KUKA KRL program: MyProgram_296().src

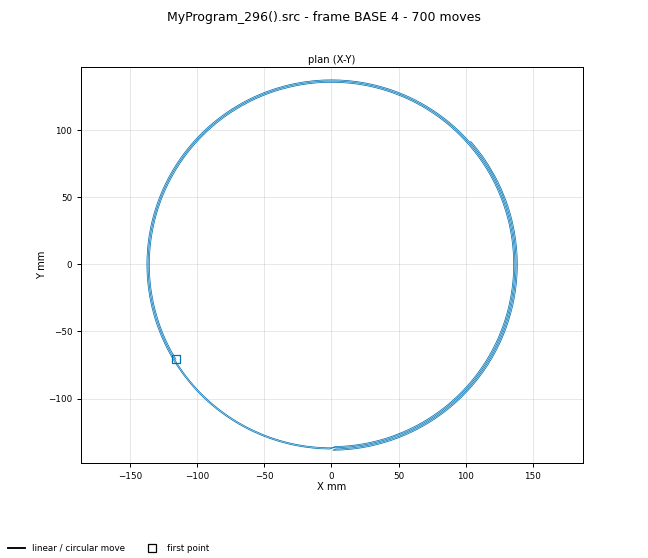
[picture p0: tool path of MyProgram_296().src in frame BASE 4, 700 of 700 moves have a stored position in this frame; points joined in program order, loops and branches not executed]
&ACCESS RVP
&REL 1
&PARAM TEMPLATE = C:\KRC\Roboter\Template\vorgabe
&PARAM EDITMASK = *
DEF MyProgram_296()
; ---- Setting reference (Base) ----
$BASE = BASE_DATA[4]

; --------------------------
; ---- Setting tool (TCP) ----
$TOOL = TOOL_DATA[3]
; --------------------------

$VEL.CP = VEL_APROX_PRINT
Startdeposition()
$VEL.CP = VEL_PRINT
LIN {X -116.0636,Y -70.6635,Z 178,A -146.1492,B 6.2959,C 0.3309,E1 6.1676,E2 238.3864} C_DIS
LIN {X -119.6803,Y -64.347,Z 178,A -149.1984,B 6.2963,C 0.3231,E1 6.1634,E2 241.4316} C_DIS
LIN {X -121.2417,Y -61.3507,Z 178,A -150.649,B 6.2965,C 0.3198,E1 6.1615,E2 242.8846} C_DIS
LIN {X -123.4162,Y -56.8493,Z 178,A -152.7977,B 6.2967,C 0.3149,E1 6.159,E2 245.0373} C_DIS
LIN {X -124.8313,Y -53.6711,Z 178,A -154.2629,B 6.2969,C 0.3111,E1 6.1573,E2 246.5015} C_DIS
LIN {X -126.1562,Y -50.4788,Z 178,A -155.7795,B 6.2971,C 0.3079,E1 6.1557,E2 248.0246} C_DIS
LIN {X -127.9876,Y -45.6377,Z 178,A -158.0309,B 6.2973,C 0.3029,E1 6.1535,E2 250.2832} C_DIS
LIN {X -129.1495,Y -42.2414,Z 178,A -159.6948,B 6.2974,C 0.3004,E1 6.152,E2 251.9649} C_DIS
LIN {X -131.3967,Y -34.6191,Z 178,A -163.2762,B 6.2978,C 0.2937,E1 6.1493,E2 255.5726} C_DIS
LIN {X -132.2272,Y -31.3001,Z 178,A -164.3938,B 6.2981,C 0.2863,E1 6.1486,E2 256.649} C_DIS
LIN {X -132.8516,Y -28.5293,Z 178,A -165.6891,B 6.2981,C 0.284,E1 6.1478,E2 257.9556} C_DIS
LIN {X -133.5646,Y -24.9844,Z 178,A -167.1822,B 6.2984,C 0.2794,E1 6.147,E2 259.4438} C_DIS
LIN {X -134.0652,Y -22.1367,Z 178,A -168.5264,B 6.2984,C 0.2773,E1 6.1464,E2 260.8025} C_DIS
LIN {X -134.7069,Y -17.8196,Z 178,A -170.3512,B 6.2987,C 0.2719,E1 6.1457,E2 262.6241} C_DIS
LIN {X -135.1168,Y -14.3862,Z 178,A -171.8433,B 6.2989,C 0.2681,E1 6.1452,E2 264.1192} C_DIS
LIN {X -135.4888,Y -10.3173,Z 178,A -173.6674,B 6.299,C 0.2643,E1 6.1448,E2 265.9546} C_DIS
LIN {X -135.7321,Y -6.3646,Z 178,A -175.3605,B 6.2992,C 0.2598,E1 6.1445,E2 267.6493} C_DIS
LIN {X -135.8577,Y -2.5014,Z 178,A -176.9735,B 6.2994,C 0.2549,E1 6.1444,E2 269.2588} C_DIS
LIN {X -135.8765,Y 1.1885,Z 178,A -178.6131,B 6.2996,C 0.2514,E1 6.1444,E2 270.9075} C_DIS
LIN {X -135.7799,Y 5.2289,Z 178,A 179.6851,B 6.2998,C 0.2464,E1 6.1445,E2 272.6076} C_DIS
LIN {X -135.6091,Y 8.5868,Z 178,A 178.1279,B 6.2998,C 0.2438,E1 6.1448,E2 274.1807} C_DIS
LIN {X -135.2372,Y 13.2071,Z 178,A 176.2276,B 6.3001,C 0.2377,E1 6.1453,E2 276.0728} C_DIS
LIN {X -134.7736,Y 17.3106,Z 178,A 174.3999,B 6.3003,C 0.2337,E1 6.1459,E2 277.9096} C_DIS
LIN {X -134.2648,Y 20.8907,Z 178,A 172.9,B 6.3004,C 0.2291,E1 6.1465,E2 279.4051} C_DIS
LIN {X -133.7038,Y 24.2246,Z 178,A 171.44,B 6.3006,C 0.2254,E1 6.1472,E2 280.8681} C_DIS
LIN {X -133.1263,Y 27.2185,Z 178,A 170.1483,B 6.3006,C 0.2218,E1 6.1479,E2 282.1594} C_DIS
LIN {X -132.3925,Y 30.5906,Z 178,A 168.6598,B 6.3008,C 0.2181,E1 6.1488,E2 283.6507} C_DIS
LIN {X -131.5728,Y 33.9457,Z 178,A 166.9358,B 6.3008,C 0.2169,E1 6.15,E2 285.4061} C_DIS
LIN {X -130.369,Y 38.3059,Z 178,A 165.1776,B 6.3011,C 0.21,E1 6.1513,E2 287.1444} C_DIS
LIN {X -129.3497,Y 41.619,Z 178,A 163.4434,B 6.3011,C 0.2089,E1 6.1528,E2 288.9105} C_DIS
LIN {X -127.4729,Y 47.0581,Z 178,A 161.2834,B 6.3014,C 0.1995,E1 6.1548,E2 291.036} C_DIS
LIN {X -125.8737,Y 51.1795,Z 178,A 159.3113,B 6.3015,C 0.1957,E1 6.1568,E2 293.0195} C_DIS
LIN {X -124.4446,Y 54.5655,Z 178,A 157.5921,B 6.3016,C 0.1934,E1 6.1587,E2 294.7579} C_DIS
LIN {X -123.226,Y 57.2606,Z 178,A 156.3891,B 6.3017,C 0.1897,E1 6.1601,E2 295.9544} C_DIS
LIN {X -121.8373,Y 60.1584,Z 178,A 154.3031,B 6.3016,C 0.1939,E1 6.1628,E2 298.1274} C_DIS
LIN {X -119.1995,Y 65.2335,Z 178,A 152.7848,B 6.3021,C 0.1784,E1 6.1647,E2 299.5357} C_DIS
LIN {X -117.7028,Y 67.897,Z 178,A 150.9757,B 6.302,C 0.1807,E1 6.1673,E2 301.4067} C_DIS
LIN {X -116.0163,Y 70.7408,Z 178,A 150.0425,B 6.3022,C 0.1724,E1 6.1685,E2 302.2829} C_DIS
LIN {X -112.7627,Y 75.8199,Z 178,A 147.1337,B 6.3022,C 0.1702,E1 6.173,E2 305.2338} C_DIS
LIN {X -110.1908,Y 79.5109,Z 178,A 145.2766,B 6.3024,C 0.1653,E1 6.176,E2 307.0844} C_DIS
LIN {X -107.6516,Y 82.9169,Z 178,A 143.3645,B 6.3024,C 0.1625,E1 6.1792,E2 309.0094} C_DIS
LIN {X -104.8415,Y 86.4421,Z 178,A 141.4392,B 6.3026,C 0.1586,E1 6.1826,E2 310.9359} C_DIS
LIN {X -101.8749,Y 89.9189,Z 178,A 139.5339,B 6.3026,C 0.1542,E1 6.1861,E2 312.8368} C_DIS
LIN {X -99.0063,Y 93.0683,Z 178,A 137.6552,B 6.3028,C 0.1513,E1 6.1897,E2 314.7239} C_DIS
LIN {X -95.9062,Y 96.2598,Z 178,A 135.7647,B 6.3028,C 0.1476,E1 6.1934,E2 316.6145} C_DIS
LIN {X -92.7534,Y 99.3014,Z 178,A 133.8742,B 6.3029,C 0.1445,E1 6.1972,E2 318.5085} C_DIS
LIN {X -89.3426,Y 102.3806,Z 178,A 131.9344,B 6.303,C 0.1408,E1 6.2013,E2 320.447} C_DIS
LIN {X -85.8899,Y 105.2941,Z 178,A 130.0021,B 6.303,C 0.1377,E1 6.2054,E2 322.3809} C_DIS
LIN {X -82.27,Y 108.1465,Z 178,A 128.0373,B 6.3031,C 0.1345,E1 6.2098,E2 324.3468} C_DIS
LIN {X -78.7448,Y 110.7397,Z 178,A 126.1286,B 6.3031,C 0.1322,E1 6.2141,E2 326.2615} C_DIS
LIN {X -74.9969,Y 113.3114,Z 178,A 123.4447,B 6.3031,C 0.1379,E1 6.2206,E2 329.0355} C_DIS
LIN {X -69.7447,Y 116.6175,Z 178,A 121.7746,B 6.3034,C 0.1231,E1 6.2243,E2 330.5904} C_DIS
LIN {X -66.8937,Y 118.2763,Z 178,A 120.1144,B 6.3034,C 0.1243,E1 6.2284,E2 332.2819} C_DIS
LIN {X -63.0682,Y 120.3568,Z 178,A 118.3471,B 6.3034,C 0.121,E1 6.2327,E2 334.0395} C_DIS
LIN {X -59.8342,Y 121.9972,Z 178,A 116.798,B 6.3034,C 0.1193,E1 6.2366,E2 335.5899} C_DIS
LIN {X -55.8012,Y 123.894,Z 178,A 114.9346,B 6.3034,C 0.1169,E1 6.2413,E2 337.45} C_DIS
LIN {X -52.2464,Y 125.434,Z 178,A 113.2307,B 6.3035,C 0.116,E1 6.2457,E2 339.1611} C_DIS
LIN {X -47.376,Y 127.3538,Z 178,A 110.5367,B 6.3035,C 0.1196,E1 6.2529,E2 341.9118} C_DIS
LIN {X -43.1002,Y 128.8635,Z 178,A 109.4047,B 6.3036,C 0.1084,E1 6.2556,E2 342.9489} C_DIS
LIN {X -38.9004,Y 130.195,Z 178,A 107.001,B 6.3036,C 0.1136,E1 6.2622,E2 345.4171} C_DIS
LIN {X -34.4811,Y 131.4335,Z 178,A 105.3513,B 6.3036,C 0.1086,E1 6.2665,E2 347.0314} C_DIS
LIN {X -31.6898,Y 132.1333,Z 178,A 104.1647,B 6.3036,C 0.1075,E1 6.2698,E2 348.214} C_DIS
LIN {X -28.623,Y 132.8313,Z 178,A 102.7874,B 6.3036,C 0.1073,E1 6.2735,E2 349.5966} C_DIS
LIN {X -25.1145,Y 133.5398,Z 178,A 101.3076,B 6.3036,C 0.1062,E1 6.2776,E2 351.0719} C_DIS
LIN {X -22.0251,Y 134.0838,Z 178,A 99.9239,B 6.3036,C 0.1063,E1 6.2814,E2 352.4622} C_DIS
LIN {X -18.0004,Y 134.6832,Z 178,A 98.1327,B 6.3036,C 0.1066,E1 6.2864,E2 354.2616} C_DIS
LIN {X -14.1094,Y 135.1465,Z 178,A 96.5823,B 6.3037,C 0.1048,E1 6.2906,E2 355.7989} C_DIS
LIN {X -10.0268,Y 135.51,Z 178,A 94.5302,B 6.3037,C 0.1087,E1 6.2965,E2 357.8889} C_DIS
LIN {X -6.7551,Y 135.7125,Z 178,A 93.4747,B 6.3037,C 0.1042,E1 6.2993,E2 358.9046} C_DIS
LIN {X -3.2262,Y 135.8433,Z 178,A 91.4247,B 6.3036,C 0.1115,E1 6.3052,E2 361.0211} C_DIS
LIN {X 1.2847,Y 135.8755,Z 178,A 89.9059,B 6.3036,C 0.1065,E1 6.3093,E2 362.4932} C_DIS
LIN {X 5.7731,Y 135.7586,Z 178,A 88.2731,B 6.3037,C 0.1033,E1 6.3138,E2 364.0939} C_DIS
LIN {X 8.3573,Y 135.6232,Z 178,A 87.0566,B 6.3037,C 0.1052,E1 6.3172,E2 365.3251} C_DIS
LIN {X 14.3269,Y 135.1231,Z 178,A 84.6214,B 6.3037,C 0.1046,E1 6.324,E2 367.7485} C_DIS
LIN {X 17.5541,Y 134.7417,Z 178,A 83.1449,B 6.3037,C 0.1066,E1 6.3281,E2 369.2373} C_DIS
LIN {X 20.9839,Y 134.2504,Z 178,A 81.677,B 6.3037,C 0.1073,E1 6.3321,E2 370.7055} C_DIS
LIN {X 25.3585,Y 133.4931,Z 178,A 79.7741,B 6.3037,C 0.1087,E1 6.3374,E2 372.6116} C_DIS
LIN {X 28.8609,Y 132.78,Z 178,A 78.3733,B 6.3037,C 0.1082,E1 6.3412,E2 373.9992} C_DIS
LIN {X 32.1612,Y 132.0196,Z 178,A 76.9512,B 6.3037,C 0.1091,E1 6.345,E2 375.4201} C_DIS
LIN {X 36.1084,Y 130.9956,Z 178,A 74.6656,B 6.3035,C 0.1184,E1 6.3514,E2 377.7734} C_DIS
LIN {X 40.7031,Y 129.6422,Z 178,A 73.2942,B 6.3035,C 0.1109,E1 6.3548,E2 379.0665} C_DIS
LIN {X 44.6522,Y 128.3339,Z 178,A 71.4391,B 6.3035,C 0.114,E1 6.3598,E2 380.9335} C_DIS
LIN {X 48.3697,Y 126.9816,Z 178,A 69.8436,B 6.3035,C 0.1146,E1 6.3639,E2 382.52} C_DIS
LIN {X 50.941,Y 125.9699,Z 178,A 68.6824,B 6.3035,C 0.1158,E1 6.3669,E2 383.6806} C_DIS
LIN {X 53.9208,Y 124.7234,Z 178,A 67.3009,B 6.3035,C 0.1176,E1 6.3705,E2 385.0643} C_DIS
LIN {X 57.2157,Y 123.2468,Z 178,A 65.8286,B 6.3035,C 0.1187,E1 6.3742,E2 386.5304} C_DIS
LIN {X 60.5933,Y 121.6227,Z 178,A 64.2467,B 6.3035,C 0.1208,E1 6.3782,E2 388.1125} C_DIS
LIN {X 64.1271,Y 119.7985,Z 178,A 62.4843,B 6.3033,C 0.1243,E1 6.3826,E2 389.8853} C_DIS
LIN {X 68.2573,Y 117.4942,Z 178,A 60.5431,B 6.3033,C 0.1263,E1 6.3873,E2 391.82} C_DIS
LIN {X 71.8437,Y 115.336,Z 178,A 58.82,B 6.3033,C 0.1284,E1 6.3914,E2 393.5381} C_DIS
LIN {X 76.4158,Y 112.3593,Z 178,A 56.6264,B 6.3033,C 0.1304,E1 6.3965,E2 395.7189} C_DIS
LIN {X 79.5335,Y 110.1744,Z 178,A 54.9237,B 6.3031,C 0.1346,E1 6.4004,E2 397.4336} C_DIS
LIN {X 83.0535,Y 107.5457,Z 178,A 53.1981,B 6.3031,C 0.1358,E1 6.4042,E2 399.144} C_DIS
LIN {X 86.2241,Y 105.021,Z 178,A 51.4142,B 6.3031,C 0.1401,E1 6.4081,E2 400.9372} C_DIS
LIN {X 89.6033,Y 102.1531,Z 178,A 49.6048,B 6.303,C 0.1426,E1 6.4119,E2 402.7398} C_DIS
LIN {X 95.2128,Y 96.9455,Z 178,A 46.5727,B 6.3029,C 0.1459,E1 6.418,E2 405.7488} C_DIS
LIN {X 99.6056,Y 92.4266,Z 178,A 43.7905,B 6.3027,C 0.1534,E1 6.4234,E2 408.547} C_DIS
LIN {X 102.5276,Y 89.1742,Z 178,A 41.9627,B 6.3027,C 0.1571,E1 6.4268,E2 410.3735} C_DIS
LIN {X 106.7379,Y 84.089,Z 178,A 39.465,B 6.3026,C 0.1587,E1 6.4312,E2 412.8371} C_DIS
LIN {X 108.7546,Y 81.4646,Z 178,A 37.8869,B 6.3024,C 0.1648,E1 6.4338,E2 414.4381} C_DIS
LIN {X 111.1727,Y 78.1318,Z 178,A 36.1359,B 6.3024,C 0.1691,E1 6.4367,E2 416.1915} C_DIS
LIN {X 113.7751,Y 74.2917,Z 178,A 34.241,B 6.3022,C 0.1727,E1 6.4396,E2 418.0797} C_DIS
LIN {X 116.1679,Y 70.491,Z 178,A 32.382,B 6.3022,C 0.1768,E1 6.4423,E2 419.9353} C_DIS
LIN {X 118.4324,Y 66.6159,Z 178,A 30.5441,B 6.302,C 0.1806,E1 6.4449,E2 421.7674} C_DIS
LIN {X 120.3327,Y 63.1142,Z 178,A 28.9081,B 6.3019,C 0.1841,E1 6.447,E2 423.3988} C_DIS
LIN {X 121.9972,Y 59.8342,Z 178,A 27.4637,B 6.3019,C 0.1863,E1 6.4488,E2 424.8309} C_DIS
LIN {X 123.6119,Y 56.4261,Z 178,A 25.7789,B 6.3017,C 0.192,E1 6.4508,E2 426.5282} C_DIS
LIN {X 126.4203,Y 49.8165,Z 178,A 23.0232,B 6.3016,C 0.1955,E1 6.4538,E2 429.252} C_DIS
LIN {X 128.0463,Y 45.4749,Z 178,A 21.0403,B 6.3014,C 0.2012,E1 6.4557,E2 431.2396} C_DIS
LIN {X 129.0556,Y 42.5232,Z 178,A 19.7314,B 6.3013,C 0.2046,E1 6.4568,E2 432.5485} C_DIS
LIN {X 129.9574,Y 39.6798,Z 178,A 18.5302,B 6.3012,C 0.2071,E1 6.4578,E2 433.7435} C_DIS
LIN {X 130.813,Y 36.7614,Z 178,A 17.2145,B 6.301,C 0.2112,E1 6.4588,E2 435.0641} C_DIS
LIN {X 131.6892,Y 33.4868,Z 178,A 15.8447,B 6.301,C 0.2141,E1 6.4598,E2 436.4274} C_DIS
LIN {X 132.6532,Y 29.4479,Z 178,A 14.0247,B 6.3007,C 0.2202,E1 6.4609,E2 438.2572} C_DIS
LIN {X 133.4336,Y 25.67,Z 178,A 12.5388,B 6.3007,C 0.2224,E1 6.4617,E2 439.7268} C_DIS
LIN {X 134.0567,Y 22.1875,Z 178,A 11.1081,B 6.3005,C 0.2255,E1 6.4624,E2 441.151} C_DIS
LIN {X 134.6366,Y 18.3559,Z 178,A 9.3768,B 6.3003,C 0.2318,E1 6.4631,E2 442.8956} C_DIS
LIN {X 135.129,Y 14.2725,Z 178,A 7.7678,B 6.3003,C 0.2346,E1 6.4636,E2 444.4903} C_DIS
LIN {X 135.5055,Y 10.0889,Z 178,A 5.5412,B 6.2997,C 0.2473,E1 6.4641,E2 446.7746} C_DIS
LIN {X 135.7694,Y 5.496,Z 178,A 3.6419,B 6.2995,C 0.2521,E1 6.4643,E2 448.6705} C_DIS
LIN {X 135.8783,Y 0.862,Z 178,A 2.2313,B 6.2997,C 0.2487,E1 6.4643,E2 450.0152} C_DIS
LIN {X 135.8374,Y -3.4376,Z 178,A -0.0974,B 6.2991,C 0.2625,E1 6.4643,E2 452.4093} C_DIS
LIN {X 135.6249,Y -8.3298,Z 178,A -1.5744,B 6.2993,C 0.2585,E1 6.464,E2 453.815} C_DIS
LIN {X 135.3457,Y -12.0589,Z 178,A -3.0356,B 6.2992,C 0.2611,E1 6.4637,E2 455.2633} C_DIS
LIN {X 134.9715,Y -15.6945,Z 178,A -4.6162,B 6.299,C 0.2662,E1 6.4632,E2 456.85} C_DIS
LIN {X 134.5126,Y -19.2305,Z 178,A -6.0496,B 6.2988,C 0.2693,E1 6.4627,E2 458.276} C_DIS
LIN {X 133.7779,Y -23.8102,Z 178,A -7.9361,B 6.2987,C 0.2736,E1 6.4618,E2 460.1554} C_DIS
LIN {X 133.1003,Y -27.3461,Z 178,A -9.4108,B 6.2985,C 0.2772,E1 6.461,E2 461.6261} C_DIS
LIN {X 132.4098,Y -30.5147,Z 178,A -10.7699,B 6.2983,C 0.2809,E1 6.4602,E2 462.9853} C_DIS
LIN {X 131.0461,Y -35.9279,Z 178,A -13.0212,B 6.2981,C 0.2858,E1 6.4586,E2 465.2259} C_DIS
LIN {X 130.2592,Y -38.6811,Z 178,A -14.2667,B 6.2979,C 0.2897,E1 6.4576,E2 466.4773} C_DIS
LIN {X 129.4087,Y -41.4344,Z 178,A -15.4712,B 6.2978,C 0.2929,E1 6.4566,E2 467.6816} C_DIS
LIN {X 127.5161,Y -46.9427,Z 178,A -17.8777,B 6.2975,C 0.2988,E1 6.4544,E2 470.0842} C_DIS
LIN {X 125.5505,Y -51.9675,Z 178,A -19.9244,B 6.2975,C 0.3011,E1 6.4523,E2 472.1041} C_DIS
LIN {X 124.5223,Y -54.3858,Z 178,A -21.2164,B 6.2971,C 0.3071,E1 6.4509,E2 473.4204} C_DIS
LIN {X 122.7582,Y -58.2572,Z 178,A -23.0205,B 6.2969,C 0.312,E1 6.4488,E2 475.2274} C_DIS
LIN {X 120.4896,Y -62.8153,Z 178,A -24.9253,B 6.2969,C 0.3135,E1 6.4464,E2 477.1037} C_DIS
LIN {X 119.1979,Y -65.2366,Z 178,A -26.2432,B 6.2965,C 0.3191,E1 6.4446,E2 478.443} C_DIS
LIN {X 116.9538,Y -69.18,Z 178,A -28.1146,B 6.2963,C 0.3233,E1 6.442,E2 480.311} C_DIS
LIN {X 114.814,Y -72.6751,Z 178,A -29.7899,B 6.2961,C 0.3267,E1 6.4395,E2 481.9811} C_DIS
LIN {X 112.3358,Y -76.4506,Z 178,A -31.681,B 6.2959,C 0.3311,E1 6.4366,E2 483.8724} C_DIS
LIN {X 109.8749,Y -79.9467,Z 178,A -33.4551,B 6.2957,C 0.3349,E1 6.4337,E2 485.6446} C_DIS
LIN {X 107.3491,Y -83.3071,Z 178,A -35.1877,B 6.2955,C 0.3384,E1 6.4308,E2 487.3737} C_DIS
LIN {X 104.5102,Y -86.8422,Z 178,A -37.0651,B 6.2953,C 0.3422,E1 6.4275,E2 489.2486} C_DIS
LIN {X 101.6631,Y -90.1586,Z 178,A -38.8818,B 6.2951,C 0.3459,E1 6.4241,E2 491.0636} C_DIS
LIN {X 98.6198,Y -93.478,Z 178,A -40.7569,B 6.2949,C 0.3496,E1 6.4206,E2 492.9374} C_DIS
LIN {X 95.4318,Y -96.7308,Z 178,A -43.1438,B 6.2943,C 0.3611,E1 6.4157,E2 495.3849} C_DIS
LIN {X 91.8687,Y -100.1198,Z 178,A -44.5572,B 6.2946,C 0.3547,E1 6.413,E2 496.7168} C_DIS
LIN {X 89.5658,Y -102.1859,Z 178,A -45.8294,B 6.2946,C 0.3568,E1 6.4104,E2 497.9861} C_DIS
LIN {X 86.7428,Y -104.5925,Z 178,A -47.5068,B 6.2942,C 0.3616,E1 6.4067,E2 499.6792} C_DIS
LIN {X 83.086,Y -107.5205,Z 178,A -49.4306,B 6.2941,C 0.3644,E1 6.4025,E2 501.5982} C_DIS
LIN {X 79.6611,Y -110.0819,Z 178,A -51.2109,B 6.2939,C 0.3673,E1 6.3985,E2 503.377} C_DIS
LIN {X 76.2647,Y -112.4616,Z 178,A -52.9478,B 6.2937,C 0.3701,E1 6.3945,E2 505.114} C_DIS
LIN {X 72.5451,Y -114.8961,Z 178,A -54.8077,B 6.2936,C 0.3729,E1 6.3902,E2 506.9736} C_DIS
LIN {X 68.5178,Y -117.3429,Z 178,A -56.7639,B 6.2934,C 0.3756,E1 6.3855,E2 508.9275} C_DIS
LIN {X 64.7472,Y -119.4648,Z 178,A -58.5983,B 6.2932,C 0.3784,E1 6.381,E2 510.7646} C_DIS
LIN {X 60.8473,Y -121.4974,Z 178,A -60.5263,B 6.293,C 0.3822,E1 6.3762,E2 512.7035} C_DIS
LIN {X 56.7439,Y -123.4649,Z 178,A -62.1933,B 6.2931,C 0.3808,E1 6.372,E2 514.3399} C_DIS
LIN {X 53.9979,Y -124.69,Z 178,A -63.73,B 6.2928,C 0.3865,E1 6.368,E2 515.9116} C_DIS
LIN {X 46.4657,Y -127.689,Z 178,A -66.7659,B 6.2928,C 0.3846,E1 6.3602,E2 518.9015} C_DIS
LIN {X 41.9034,Y -129.2588,Z 178,A -68.7651,B 6.2928,C 0.3862,E1 6.3549,E2 520.8976} C_DIS
LIN {X 38.4539,Y -130.3257,Z 178,A -70.4167,B 6.2926,C 0.3896,E1 6.3505,E2 522.5667} C_DIS
LIN {X 34.8173,Y -131.3439,Z 178,A -71.9768,B 6.2926,C 0.3905,E1 6.3463,E2 524.1237} C_DIS
LIN {X 31.4044,Y -132.2021,Z 178,A -73.3966,B 6.2925,C 0.3907,E1 6.3424,E2 525.5364} C_DIS
LIN {X 28.2597,Y -132.9098,Z 178,A -74.9104,B 6.2923,C 0.394,E1 6.3383,E2 527.0707} C_DIS
LIN {X 24.0792,Y -133.7298,Z 178,A -76.8012,B 6.2921,C 0.3965,E1 6.333,E2 528.9745} C_DIS
LIN {X 18.4191,Y -134.6284,Z 178,A -78.9444,B 6.2923,C 0.3939,E1 6.3272,E2 531.0846} C_DIS
LIN {X 15.1531,Y -135.0342,Z 178,A -81.1475,B 6.2915,C 0.4061,E1 6.3208,E2 533.3915} C_DIS
LIN {X 9.2312,Y -135.5681,Z 178,A -82.7583,B 6.2923,C 0.3943,E1 6.3166,E2 534.8903} C_DIS
LIN {X 2.4002,Y -135.8594,Z 178,A -85.6824,B 6.2922,C 0.3955,E1 6.3085,E2 537.8211} C_DIS
LIN {X 2.4002,Y -135.8594,Z 178,A -85.6824,B 6.2922,C 0.3955,E1 6.3085,E2 537.8212} C_DIS
Enddeposition()
LIN {X 0.9937,Y -136.781,Z 178,A -85.9393,B 6.2292,C 0.3941,E1 6.2447,E2 538.0864} C_DIS
Startdeposition()
$VEL.CP = VEL_PRINT
LIN {X 7.0143,Y -136.6048,Z 178,A -83.1394,B 6.2294,C 0.3897,E1 6.2526,E2 535.2495} C_DIS
LIN {X 13.8862,Y -136.08,Z 178,A -80.1066,B 6.2296,C 0.3865,E1 6.2611,E2 532.1964} C_DIS
LIN {X 22.8856,Y -134.857,Z 178,A -76.3832,B 6.2296,C 0.3857,E1 6.2714,E2 528.4815} C_DIS
LIN {X 26.6198,Y -134.1709,Z 178,A -74.7602,B 6.2298,C 0.3842,E1 6.2758,E2 526.8533} C_DIS
LIN {X 30.257,Y -133.3962,Z 178,A -73.3123,B 6.2298,C 0.3847,E1 6.2797,E2 525.4186} C_DIS
LIN {X 33.2653,Y -132.6783,Z 178,A -71.9723,B 6.2298,C 0.383,E1 6.2834,E2 524.072} C_DIS
LIN {X 37.0999,Y -131.6573,Z 178,A -70.408,B 6.2298,C 0.383,E1 6.2876,E2 522.5193} C_DIS
LIN {X 40.7775,Y -130.5671,Z 178,A -68.7967,B 6.2299,C 0.3814,E1 6.2919,E2 520.9063} C_DIS
LIN {X 43.894,Y -129.5522,Z 178,A -67.2601,B 6.2302,C 0.3775,E1 6.296,E2 519.3475} C_DIS
LIN {X 53.8396,Y -125.7436,Z 178,A -63.1247,B 6.2302,C 0.3775,E1 6.3067,E2 515.2513} C_DIS
LIN {X 58.4249,Y -123.6802,Z 178,A -61.0159,B 6.2304,C 0.3747,E1 6.312,E2 513.1408} C_DIS
LIN {X 61.008,Y -122.4265,Z 178,A -59.7426,B 6.2305,C 0.3719,E1 6.3153,E2 511.8574} C_DIS
LIN {X 64.4799,Y -120.6354,Z 178,A -57.9955,B 6.2308,C 0.3678,E1 6.3196,E2 510.0947} C_DIS
LIN {X 68.4273,Y -118.4406,Z 178,A -56.1417,B 6.2308,C 0.3656,E1 6.3241,E2 508.2443} C_DIS
LIN {X 72.5143,Y -115.9837,Z 178,A -54.1992,B 6.231,C 0.3633,E1 6.3287,E2 506.3072} C_DIS
LIN {X 76.1478,Y -113.6311,Z 178,A -52.4262,B 6.2312,C 0.3609,E1 6.3328,E2 504.538} C_DIS
LIN {X 79.823,Y -111.0804,Z 178,A -50.5401,B 6.2314,C 0.3574,E1 6.3372,E2 502.6487} C_DIS
LIN {X 83.246,Y -108.5385,Z 178,A -48.8043,B 6.2314,C 0.355,E1 6.341,E2 500.9178} C_DIS
LIN {X 86.8047,Y -105.7143,Z 178,A -46.9088,B 6.2317,C 0.3516,E1 6.3451,E2 499.0216} C_DIS
LIN {X 91.8683,Y -101.3444,Z 178,A -43.8168,B 6.2323,C 0.3413,E1 6.3517,E2 495.8894} C_DIS
LIN {X 94.8582,Y -98.552,Z 178,A -42.3552,B 6.2323,C 0.3419,E1 6.3546,E2 494.4592} C_DIS
LIN {X 98.5146,Y -94.897,Z 178,A -40.3012,B 6.2323,C 0.3392,E1 6.3586,E2 492.4177} C_DIS
LIN {X 101.6106,Y -91.5747,Z 178,A -38.4541,B 6.2326,C 0.3359,E1 6.362,E2 490.576} C_DIS
LIN {X 104.4722,Y -88.2959,Z 178,A -36.6477,B 6.2328,C 0.3321,E1 6.3653,E2 488.77} C_DIS
LIN {X 107.3567,Y -84.765,Z 178,A -34.7947,B 6.2329,C 0.3287,E1 6.3685,E2 486.9226} C_DIS
LIN {X 109.9748,Y -81.3399,Z 178,A -33.0306,B 6.2331,C 0.3252,E1 6.3715,E2 485.1622} C_DIS
LIN {X 112.4928,Y -77.8201,Z 178,A -31.2377,B 6.2333,C 0.3211,E1 6.3744,E2 483.3703} C_DIS
LIN {X 114.9924,Y -74.0767,Z 178,A -29.3673,B 6.2336,C 0.3168,E1 6.3772,E2 481.5} C_DIS
LIN {X 117.4366,Y -70.1364,Z 178,A -27.5436,B 6.2336,C 0.3139,E1 6.3799,E2 479.6897} C_DIS
LIN {X 119.4847,Y -66.5884,Z 178,A -25.963,B 6.2338,C 0.3119,E1 6.382,E2 478.1251} C_DIS
LIN {X 121.8235,Y -62.2011,Z 178,A -23.8208,B 6.2341,C 0.3055,E1 6.3848,E2 475.9732} C_DIS
LIN {X 123.4477,Y -58.9116,Z 178,A -22.2217,B 6.2344,C 0.3004,E1 6.3868,E2 474.3646} C_DIS
LIN {X 125.4043,Y -54.6243,Z 178,A -20.512,B 6.2344,C 0.2997,E1 6.3887,E2 472.6871} C_DIS
LIN {X 126.7997,Y -51.3009,Z 178,A -19.122,B 6.2344,C 0.2976,E1 6.3902,E2 471.311} C_DIS
LIN {X 127.9897,Y -48.2561,Z 178,A -17.6236,B 6.2348,C 0.2918,E1 6.3917,E2 469.7949} C_DIS
LIN {X 129.3482,Y -44.4871,Z 178,A -16.0266,B 6.2349,C 0.2886,E1 6.3932,E2 468.2067} C_DIS
LIN {X 130.4059,Y -41.284,Z 178,A -14.586,B 6.2351,C 0.2842,E1 6.3944,E2 466.7613} C_DIS
LIN {X 131.3176,Y -38.284,Z 178,A -13.3802,B 6.2351,C 0.2824,E1 6.3954,E2 465.5681} C_DIS
LIN {X 132.0354,Y -35.7334,Z 178,A -12.3491,B 6.2353,C 0.2807,E1 6.3961,E2 464.5461} C_DIS
LIN {X 132.8418,Y -32.6091,Z 178,A -10.9141,B 6.2355,C 0.2755,E1 6.3971,E2 463.0993} C_DIS
LIN {X 133.6585,Y -29.0765,Z 178,A -9.3989,B 6.2357,C 0.2713,E1 6.398,E2 461.5831} C_DIS
LIN {X 134.3139,Y -25.8806,Z 178,A -8.0398,B 6.2358,C 0.2675,E1 6.3988,E2 460.2238} C_DIS
LIN {X 134.9897,Y -22.0897,Z 178,A -6.4213,B 6.236,C 0.2629,E1 6.3995,E2 458.6032} C_DIS
LIN {X 135.5908,Y -18.0342,Z 178,A -4.811,B 6.2362,C 0.2598,E1 6.4001,E2 457.0051} C_DIS
LIN {X 136.0879,Y -13.8085,Z 178,A -2.5856,B 6.2367,C 0.2472,E1 6.4008,E2 454.7215} C_DIS
LIN {X 136.4609,Y -9.4217,Z 178,A -0.6421,B 6.237,C 0.2402,E1 6.4012,E2 452.7637} C_DIS
LIN {X 136.7206,Y -4.2081,Z 178,A 0.9836,B 6.2368,C 0.2435,E1 6.4013,E2 451.2081} C_DIS
LIN {X 136.7815,Y -1.0613,Z 178,A 2.9325,B 6.2374,C 0.229,E1 6.4013,E2 449.1773} C_DIS
LIN {X 136.6944,Y 4.9829,Z 178,A 4.802,B 6.2372,C 0.2331,E1 6.4013,E2 447.3908} C_DIS
LIN {X 136.3411,Y 11.0178,Z 178,A 7.1487,B 6.2374,C 0.229,E1 6.4008,E2 445.0659} C_DIS
LIN {X 135.7969,Y 16.4097,Z 178,A 9.3818,B 6.2376,C 0.2232,E1 6.4001,E2 442.8357} C_DIS
LIN {X 135.2647,Y 20.3425,Z 178,A 10.8423,B 6.2376,C 0.2219,E1 6.3995,E2 441.3996} C_DIS
LIN {X 134.696,Y 23.8134,Z 178,A 12.3983,B 6.2378,C 0.2163,E1 6.3988,E2 439.8321} C_DIS
LIN {X 134.0427,Y 27.2495,Z 178,A 13.7971,B 6.2379,C 0.2133,E1 6.398,E2 438.4406} C_DIS
LIN {X 133.423,Y 30.1393,Z 178,A 14.9502,B 6.238,C 0.2113,E1 6.3974,E2 437.2974} C_DIS
LIN {X 132.7895,Y 32.8261,Z 178,A 16.2855,B 6.2382,C 0.2051,E1 6.3965,E2 435.9388} C_DIS
LIN {X 131.8515,Y 36.4054,Z 178,A 17.7044,B 6.2382,C 0.203,E1 6.3954,E2 434.5354} C_DIS
LIN {X 130.8627,Y 39.8115,Z 178,A 18.9442,B 6.2382,C 0.203,E1 6.3945,E2 433.3256} C_DIS
LIN {X 129.8964,Y 42.8604,Z 178,A 20.4036,B 6.2385,C 0.1974,E1 6.3932,E2 431.8503} C_DIS
LIN {X 128.8212,Y 45.9916,Z 178,A 21.8189,B 6.2385,C 0.1932,E1 6.3919,E2 430.4306} C_DIS
LIN {X 127.7315,Y 48.9392,Z 178,A 23.0076,B 6.2386,C 0.1918,E1 6.3907,E2 429.2572} C_DIS
LIN {X 126.476,Y 52.0979,Z 178,A 24.731,B 6.2389,C 0.1831,E1 6.3889,E2 427.4953} C_DIS
LIN {X 125.2112,Y 55.0709,Z 178,A 25.9385,B 6.2389,C 0.182,E1 6.3876,E2 426.3055} C_DIS
LIN {X 123.6218,Y 58.5471,Z 178,A 27.4571,B 6.239,C 0.1792,E1 6.3858,E2 424.7963} C_DIS
LIN {X 122.0165,Y 61.8218,Z 178,A 28.8945,B 6.239,C 0.1768,E1 6.384,E2 423.3695} C_DIS
LIN {X 120.2231,Y 65.2454,Z 178,A 30.5035,B 6.2392,C 0.1729,E1 6.3819,E2 421.761} C_DIS
LIN {X 118.211,Y 68.824,Z 178,A 32.2071,B 6.2392,C 0.1689,E1 6.3795,E2 420.0586} C_DIS
LIN {X 115.9754,Y 72.5277,Z 178,A 34.0126,B 6.2394,C 0.1646,E1 6.3769,E2 418.2531} C_DIS
LIN {X 113.5789,Y 76.226,Z 178,A 35.8177,B 6.2394,C 0.1609,E1 6.3741,E2 416.4524} C_DIS
LIN {X 111.0987,Y 79.7974,Z 178,A 37.6117,B 6.2396,C 0.1571,E1 6.3712,E2 414.6611} C_DIS
LIN {X 108.6744,Y 83.0683,Z 178,A 39.242,B 6.2396,C 0.1544,E1 6.3685,E2 413.0396} C_DIS
LIN {X 106.5603,Y 85.7635,Z 178,A 40.7585,B 6.2398,C 0.1499,E1 6.3658,E2 411.5123} C_DIS
LIN {X 103.3768,Y 89.5759,Z 178,A 42.7564,B 6.2398,C 0.1467,E1 6.3622,E2 409.5242} C_DIS
LIN {X 100.5575,Y 92.7292,Z 178,A 44.6373,B 6.24,C 0.1412,E1 6.3586,E2 407.6291} C_DIS
LIN {X 96.7471,Y 96.6986,Z 178,A 46.7218,B 6.24,C 0.1399,E1 6.3546,E2 405.5716} C_DIS
LIN {X 92.7195,Y 100.5663,Z 178,A 49.0276,B 6.24,C 0.1359,E1 6.35,E2 403.2694} C_DIS
LIN {X 89.4084,Y 103.5212,Z 178,A 50.8664,B 6.2402,C 0.1327,E1 6.3461,E2 401.4328} C_DIS
LIN {X 86.0779,Y 106.3068,Z 178,A 52.6024,B 6.2402,C 0.1306,E1 6.3424,E2 399.7068} C_DIS
LIN {X 82.8994,Y 108.8035,Z 178,A 54.3427,B 6.2402,C 0.1269,E1 6.3385,E2 397.9604} C_DIS
LIN {X 79.5471,Y 111.2777,Z 178,A 56.0168,B 6.2403,C 0.1251,E1 6.3348,E2 396.2949} C_DIS
LIN {X 76.0397,Y 113.7033,Z 178,A 57.8094,B 6.2403,C 0.1221,E1 6.3306,E2 394.5014} C_DIS
LIN {X 72.2393,Y 116.1548,Z 178,A 59.6747,B 6.2404,C 0.1196,E1 6.3262,E2 392.6396} C_DIS
LIN {X 68.3691,Y 118.4743,Z 178,A 61.5347,B 6.2404,C 0.1173,E1 6.3217,E2 390.7833} C_DIS
LIN {X 64.5467,Y 120.5995,Z 178,A 63.3359,B 6.2405,C 0.1152,E1 6.3173,E2 388.9859} C_DIS
LIN {X 61.2122,Y 122.3257,Z 178,A 64.799,B 6.2405,C 0.1148,E1 6.3137,E2 387.5364} C_DIS
LIN {X 57.849,Y 123.9502,Z 178,A 66.4324,B 6.2405,C 0.1119,E1 6.3096,E2 385.8946} C_DIS
LIN {X 54.465,Y 125.4732,Z 178,A 67.911,B 6.2405,C 0.1111,E1 6.3058,E2 384.4254} C_DIS
LIN {X 51.309,Y 126.7965,Z 178,A 69.2894,B 6.2405,C 0.1104,E1 6.3023,E2 383.054} C_DIS
LIN {X 48.619,Y 127.8538,Z 178,A 70.4732,B 6.2406,C 0.1095,E1 6.2992,E2 381.8737} C_DIS
LIN {X 45.2143,Y 129.0961,Z 178,A 72.0325,B 6.2406,C 0.1074,E1 6.2951,E2 380.3096} C_DIS
LIN {X 42.2972,Y 130.0823,Z 178,A 73.4587,B 6.2406,C 0.1043,E1 6.2913,E2 378.8668} C_DIS
LIN {X 37.8153,Y 131.4548,Z 178,A 75.4038,B 6.2407,C 0.1029,E1 6.2861,E2 376.9243} C_DIS
LIN {X 33.6513,Y 132.5804,Z 178,A 77.1027,B 6.2407,C 0.1031,E1 6.2815,E2 375.2391} C_DIS
LIN {X 29.6954,Y 133.5244,Z 178,A 78.7725,B 6.2407,C 0.1024,E1 6.277,E2 373.574} C_DIS
LIN {X 25.8451,Y 134.3207,Z 178,A 80.416,B 6.2407,C 0.1015,E1 6.2725,E2 371.9313} C_DIS
LIN {X 22.4458,Y 134.9303,Z 178,A 81.8522,B 6.2407,C 0.1009,E1 6.2685,E2 370.4969} C_DIS
LIN {X 18.702,Y 135.5016,Z 178,A 83.7273,B 6.2408,C 0.0963,E1 6.2633,E2 368.5867} C_DIS
LIN {X 15.3526,Y 135.9222,Z 178,A 85.2227,B 6.2408,C 0.0946,E1 6.2591,E2 367.0817} C_DIS
LIN {X 11.697,Y 136.2837,Z 178,A 86.5157,B 6.2408,C 0.0976,E1 6.2556,E2 365.8196} C_DIS
LIN {X 8.0217,Y 136.5498,Z 178,A 88.4945,B 6.2408,C 0.0914,E1 6.2499,E2 363.7876} C_DIS
LIN {X 3.1021,Y 136.7513,Z 178,A 89.9166,B 6.2408,C 0.0998,E1 6.2462,E2 362.4455} C_DIS
LIN {X -3.9297,Y 136.7283,Z 178,A 92.8771,B 6.2408,C 0.0997,E1 6.2379,E2 359.4846} C_DIS
LIN {X -6.5681,Y 136.6272,Z 178,A 94.6736,B 6.2409,C 0.0906,E1 6.2327,E2 357.6035} C_DIS
LIN {X -11.7409,Y 136.28,Z 178,A 96.1523,B 6.2408,C 0.1002,E1 6.2288,E2 356.2114} C_DIS
LIN {X -15.1734,Y 135.9415,Z 178,A 97.6966,B 6.2408,C 0.0993,E1 6.2244,E2 354.6557} C_DIS
LIN {X -19.1134,Y 135.4428,Z 178,A 99.3372,B 6.2408,C 0.1002,E1 6.2199,E2 353.0189} C_DIS
LIN {X -22.0645,Y 134.994,Z 178,A 100.4539,B 6.2408,C 0.1025,E1 6.2169,E2 351.9192} C_DIS
LIN {X -25.578,Y 134.3718,Z 178,A 102.0512,B 6.2408,C 0.1019,E1 6.2125,E2 350.3102} C_DIS
LIN {X -28.4393,Y 133.7961,Z 178,A 103.263,B 6.2408,C 0.1027,E1 6.2091,E2 349.1005} C_DIS
LIN {X -31.8302,Y 133.0296,Z 178,A 104.7985,B 6.2408,C 0.1027,E1 6.2049,E2 347.5561} C_DIS
LIN {X -35.2494,Y 132.1645,Z 178,A 106.2329,B 6.2407,C 0.1042,E1 6.2011,E2 346.1279} C_DIS
LIN {X -38.7487,Y 131.1816,Z 178,A 107.7775,B 6.2407,C 0.1051,E1 6.1969,E2 344.5816} C_DIS
LIN {X -42.5857,Y 129.9879,Z 178,A 109.4039,B 6.2407,C 0.1072,E1 6.1926,E2 342.9633} C_DIS
LIN {X -48.8812,Y 127.754,Z 178,A 112.3044,B 6.2407,C 0.1087,E1 6.185,E2 340.0523} C_DIS
LIN {X -53.8752,Y 125.7282,Z 178,A 114.5788,B 6.2406,C 0.1109,E1 6.1791,E2 337.7774} C_DIS
LIN {X -57.0897,Y 124.3012,Z 178,A 116.0319,B 6.2406,C 0.1128,E1 6.1754,E2 336.3278} C_DIS
LIN {X -59.6197,Y 123.1094,Z 178,A 117.22,B 6.2406,C 0.114,E1 6.1724,E2 335.1386} C_DIS
LIN {X -62.5654,Y 121.638,Z 178,A 118.7491,B 6.2406,C 0.114,E1 6.1686,E2 333.5922} C_DIS
LIN {X -66.6785,Y 119.4345,Z 178,A 120.7509,B 6.2405,C 0.1161,E1 6.1637,E2 331.5861} C_DIS
LIN {X -70.6221,Y 117.1453,Z 178,A 122.4027,B 6.2404,C 0.1219,E1 6.1598,E2 329.9675} C_DIS
LIN {X -74.0479,Y 115.0109,Z 178,A 124.3574,B 6.2404,C 0.1214,E1 6.1551,E2 327.9817} C_DIS
LIN {X -77.6386,Y 112.6179,Z 178,A 126.1934,B 6.2404,C 0.1239,E1 6.1508,E2 326.1437} C_DIS
LIN {X -81.3667,Y 109.9549,Z 178,A 128.1314,B 6.2403,C 0.1269,E1 6.1464,E2 324.205} C_DIS
LIN {X -84.8917,Y 107.2567,Z 178,A 130.0542,B 6.2403,C 0.1295,E1 6.1422,E2 322.2759} C_DIS
LIN {X -88.4302,Y 104.358,Z 178,A 131.9804,B 6.2402,C 0.1328,E1 6.1381,E2 320.3501} C_DIS
LIN {X -91.519,Y 101.6604,Z 178,A 133.7044,B 6.2401,C 0.136,E1 6.1345,E2 318.6268} C_DIS
LIN {X -94.6574,Y 98.7445,Z 178,A 135.5235,B 6.2401,C 0.1393,E1 6.1308,E2 316.8062} C_DIS
LIN {X -97.8767,Y 95.5547,Z 178,A 137.4689,B 6.2399,C 0.1426,E1 6.1269,E2 314.8567} C_DIS
LIN {X -100.9463,Y 92.3062,Z 178,A 139.4094,B 6.2399,C 0.1457,E1 6.1232,E2 312.9094} C_DIS
LIN {X -103.9386,Y 88.9236,Z 178,A 141.34,B 6.2398,C 0.1494,E1 6.1197,E2 310.9757} C_DIS
LIN {X -106.8754,Y 85.3708,Z 178,A 143.2818,B 6.2397,C 0.1536,E1 6.1163,E2 309.0342} C_DIS
LIN {X -109.6543,Y 81.7704,Z 178,A 145.1547,B 6.2396,C 0.1583,E1 6.1131,E2 307.167} C_DIS
LIN {X -112.0886,Y 78.401,Z 178,A 147.0064,B 6.2395,C 0.1611,E1 6.1101,E2 305.3032} C_DIS
LIN {X -113.7953,Y 75.9018,Z 178,A 148.3277,B 6.2395,C 0.1635,E1 6.1081,E2 303.9765} C_DIS
LIN {X -116.995,Y 70.8706,Z 178,A 150.7809,B 6.2393,C 0.1701,E1 6.1044,E2 301.5311} C_DIS
LIN {X -119.1541,Y 67.1773,Z 178,A 152.6196,B 6.2391,C 0.1741,E1 6.1019,E2 299.6882} C_DIS
LIN {X -120.8566,Y 64.0613,Z 178,A 154.4391,B 6.2391,C 0.1742,E1 6.0994,E2 297.8287} C_DIS
LIN {X -122.5022,Y 60.8543,Z 178,A 155.4993,B 6.2389,C 0.1829,E1 6.0982,E2 296.8257} C_DIS
LIN {X -123.7079,Y 58.367,Z 178,A 156.7886,B 6.2389,C 0.1845,E1 6.0966,E2 295.5213} C_DIS
LIN {X -125.3432,Y 54.7656,Z 178,A 158.5391,B 6.2387,C 0.1879,E1 6.0946,E2 293.7606} C_DIS
LIN {X -126.5992,Y 51.7985,Z 178,A 159.8141,B 6.2387,C 0.1922,E1 6.0932,E2 292.4961} C_DIS
LIN {X -127.9131,Y 48.4607,Z 178,A 161.2753,B 6.2385,C 0.1967,E1 6.0918,E2 291.0414} C_DIS
LIN {X -130.2347,Y 41.8201,Z 178,A 164.3784,B 6.2383,C 0.203,E1 6.089,E2 287.9217} C_DIS
LIN {X -131.9797,Y 35.9422,Z 178,A 166.9968,B 6.2381,C 0.2096,E1 6.0869,E2 285.2994} C_DIS
LIN {X -132.8936,Y 32.3943,Z 178,A 168.6591,B 6.238,C 0.2125,E1 6.0858,E2 283.6226} C_DIS
LIN {X -133.6839,Y 28.9586,Z 178,A 170.0332,B 6.2378,C 0.2177,E1 6.0849,E2 282.2626} C_DIS
LIN {X -134.2239,Y 26.3515,Z 178,A 171.4147,B 6.2378,C 0.2181,E1 6.0842,E2 280.8489} C_DIS
LIN {X -135.0172,Y 21.925,Z 178,A 173.3235,B 6.2376,C 0.2231,E1 6.0833,E2 278.9386} C_DIS
LIN {X -135.598,Y 17.9788,Z 178,A 174.9217,B 6.2374,C 0.2286,E1 6.0827,E2 277.3508} C_DIS
LIN {X -136.0136,Y 14.5032,Z 178,A 176.4892,B 6.2373,C 0.2317,E1 6.0822,E2 275.7718} C_DIS
LIN {X -136.3665,Y 10.7137,Z 178,A 178.2316,B 6.2372,C 0.2347,E1 6.0818,E2 274.0123} C_DIS
LIN {X -136.6496,Y 6.1225,Z 178,A -179.858,B 6.237,C 0.2404,E1 6.0815,E2 272.1056} C_DIS
LIN {X -136.7672,Y 2.1942,Z 178,A -178.2559,B 6.2368,C 0.2456,E1 6.0814,E2 270.5103} C_DIS
LIN {X -136.7725,Y -1.8726,Z 178,A -176.6504,B 6.2365,C 0.2515,E1 6.0814,E2 268.9184} C_DIS
LIN {X -136.676,Y -5.4545,Z 178,A -174.9356,B 6.2365,C 0.2535,E1 6.0816,E2 267.178} C_DIS
LIN {X -136.4421,Y -9.6792,Z 178,A -173.2043,B 6.2362,C 0.259,E1 6.0819,E2 265.4531} C_DIS
LIN {X -136.1497,Y -13.1643,Z 178,A -171.6589,B 6.2361,C 0.2623,E1 6.0823,E2 263.8987} C_DIS
LIN {X -135.7191,Y -17.0552,Z 178,A -169.8919,B 6.2359,C 0.2656,E1 6.0828,E2 262.117} C_DIS
LIN {X -135.1763,Y -20.9137,Z 178,A -168.3506,B 6.2357,C 0.2712,E1 6.0835,E2 260.5883} C_DIS
LIN {X -134.6008,Y -24.345,Z 178,A -166.8199,B 6.2356,C 0.2745,E1 6.0842,E2 259.0494} C_DIS
LIN {X -133.7975,Y -28.4328,Z 178,A -165.1869,B 6.2353,C 0.2805,E1 6.0851,E2 257.4317} C_DIS
LIN {X -133.0693,Y -31.6653,Z 178,A -163.5422,B 6.2353,C 0.2816,E1 6.0862,E2 255.7555} C_DIS
LIN {X -130.8679,Y -39.7945,Z 178,A -160.062,B 6.2348,C 0.2918,E1 6.0888,E2 252.2838} C_DIS
LIN {X -129.6789,Y -43.5137,Z 178,A -157.8108,B 6.2348,C 0.2895,E1 6.0908,E2 249.9554} C_DIS
LIN {X -128.1288,Y -47.8847,Z 178,A -156.4749,B 6.2343,C 0.3013,E1 6.092,E2 248.6979} C_DIS
LIN {X -127.1483,Y -50.4361,Z 178,A -155.2531,B 6.2343,C 0.3035,E1 6.0933,E2 247.467} C_DIS
LIN {X -125.6947,Y -53.9528,Z 178,A -153.5692,B 6.2341,C 0.3067,E1 6.0951,E2 245.7725} C_DIS
LIN {X -124.3042,Y -57.0833,Z 178,A -152.0708,B 6.2339,C 0.3097,E1 6.0969,E2 244.2668} C_DIS
LIN {X -122.496,Y -60.867,Z 178,A -150.3038,B 6.2337,C 0.314,E1 6.099,E2 242.4994} C_DIS
LIN {X -120.4756,Y -64.7773,Z 178,A -148.4031,B 6.2335,C 0.318,E1 6.1015,E2 240.5925} C_DIS
LIN {X -118.1137,Y -68.9909,Z 178,A -146.2502,B 6.2333,C 0.3215,E1 6.1045,E2 238.4241} C_DIS
LIN {X -115.7426,Y -72.8981,Z 178,A -144.367,B 6.2331,C 0.3264,E1 6.1073,E2 236.5457} C_DIS
LIN {X -113.243,Y -76.7235,Z 178,A -142.3815,B 6.2329,C 0.33,E1 6.1103,E2 234.5518} C_DIS
LIN {X -110.5695,Y -80.5291,Z 178,A -140.5964,B 6.2325,C 0.3363,E1 6.1132,E2 232.7884} C_DIS
LIN {X -108.2177,Y -83.6626,Z 178,A -138.7385,B 6.2325,C 0.3375,E1 6.1164,E2 230.9033} C_DIS
LIN {X -105.5435,Y -87.0122,Z 178,A -136.8625,B 6.2323,C 0.3404,E1 6.1197,E2 229.0177} C_DIS
LIN {X -102.6501,Y -90.4073,Z 178,A -134.5418,B 6.2323,C 0.3391,E1 6.1241,E2 226.6393} C_DIS
LIN {X -99.5507,Y -93.809,Z 178,A -133.0379,B 6.2319,C 0.3479,E1 6.1269,E2 225.1905} C_DIS
LIN {X -97.2525,Y -96.1899,Z 178,A -131.6169,B 6.2318,C 0.3502,E1 6.1296,E2 223.7654} C_DIS
LIN {X -94.1487,Y -99.2302,Z 178,A -129.7763,B 6.2316,C 0.3535,E1 6.1333,E2 221.9225} C_DIS
LIN {X -90.9159,Y -102.2004,Z 178,A -127.869,B 6.2314,C 0.356,E1 6.1373,E2 220.0069} C_DIS
LIN {X -87.6867,Y -104.9838,Z 178,A -126.0865,B 6.2313,C 0.3592,E1 6.1411,E2 218.2251} C_DIS
LIN {X -84.1434,Y -107.845,Z 178,A -124.1493,B 6.2311,C 0.3621,E1 6.1454,E2 216.2844} C_DIS
LIN {X -80.8573,Y -110.3294,Z 178,A -122.4746,B 6.2309,C 0.3655,E1 6.1491,E2 214.6163} C_DIS
LIN {X -77.2899,Y -112.8572,Z 178,A -120.5672,B 6.2308,C 0.3674,E1 6.1535,E2 212.6993} C_DIS
LIN {X -73.5506,Y -115.3292,Z 178,A -118.7325,B 6.2306,C 0.3707,E1 6.1578,E2 210.8702} C_DIS
LIN {X -70.1207,Y -117.446,Z 178,A -116.9537,B 6.2306,C 0.3719,E1 6.1621,E2 209.0798} C_DIS
LIN {X -66.1746,Y -119.7138,Z 178,A -115.0682,B 6.2304,C 0.3747,E1 6.1666,E2 207.1969} C_DIS
LIN {X -62.3866,Y -121.729,Z 178,A -113.2249,B 6.2303,C 0.3763,E1 6.1712,E2 205.3475} C_DIS
LIN {X -59.1175,Y -123.3493,Z 178,A -111.7763,B 6.2301,C 0.379,E1 6.1748,E2 203.9091} C_DIS
LIN {X -56.0351,Y -124.7799,Z 178,A -110.3652,B 6.23,C 0.3807,E1 6.1784,E2 202.4995} C_DIS
LIN {X -53.0109,Y -126.0947,Z 178,A -109.0394,B 6.2299,C 0.3829,E1 6.1818,E2 201.1808} C_DIS
LIN {X -50.4859,Y -127.1283,Z 178,A -107.6379,B 6.2299,C 0.3806,E1 6.1855,E2 199.7457} C_DIS
LIN {X -46.7867,Y -128.5345,Z 178,A -106.2564,B 6.2297,C 0.3857,E1 6.189,E2 198.3996} C_DIS
LIN {X -43.5841,Y -129.6554,Z 178,A -104.5132,B 6.2299,C 0.3826,E1 6.1938,E2 196.6145} C_DIS
LIN {X -38.8046,Y -131.1652,Z 178,A -102.499,B 6.2297,C 0.3853,E1 6.1991,E2 194.6109} C_DIS
LIN {X -35.2878,Y -132.1542,Z 178,A -101.0651,B 6.2296,C 0.3875,E1 6.2029,E2 193.1891} C_DIS
LIN {X -32.5097,Y -132.8658,Z 178,A -99.9025,B 6.2295,C 0.3887,E1 6.2061,E2 192.0313} C_DIS
LIN {X -29.8238,Y -133.4951,Z 178,A -98.528,B 6.2296,C 0.3864,E1 6.2099,E2 190.6281} C_DIS
LIN {X -25.9115,Y -134.308,Z 178,A -96.9813,B 6.2295,C 0.3888,E1 6.2141,E2 189.0973} C_DIS
LIN {X -21.8121,Y -135.0361,Z 178,A -94.88,B 6.2298,C 0.3846,E1 6.22,E2 186.9491} C_DIS
LIN {X -18.2992,Y -135.556,Z 178,A -93.1162,B 6.23,C 0.3811,E1 6.225,E2 185.1487} C_DIS
LIN {X -13.2943,Y -136.1372,Z 178,A -91.8632,B 6.2292,C 0.3934,E1 6.2282,E2 184.0064} C_DIS
LIN {X -7.4064,Y -136.5851,Z 178,A -89.0276,B 6.2295,C 0.3886,E1 6.2362,E2 181.123} C_DIS
LIN {X -3.4054,Y -136.7429,Z 178,A -87.3786,B 6.2295,C 0.3889,E1 6.2408,E2 179.477} C_DIS
LIN {X 0.9937,Y -136.781,Z 178,A -85.937,B 6.2291,C 0.3944,E1 6.2447,E2 178.0864} C_DIS
Enddeposition()
LIN {X 0.9937,Y -136.781,Z 178,A -85.937,B 6.2291,C 0.3944,E1 6.2447,E2 178.0864} C_DIS
Startdeposition()
$VEL.CP = VEL_PRINT
LIN {X -1.1234,Y -137.6849,Z 178,A -87.0809,B 6.1678,C 0.4013,E1 6.1805,E2 179.3151} C_DIS
LIN {X -4.5941,Y -137.6145,Z 178,A -88.5059,B 6.1678,C 0.4011,E1 6.1765,E2 180.7383} C_DIS
LIN {X -7.5479,Y -137.4834,Z 178,A -89.7432,B 6.1678,C 0.4011,E1 6.173,E2 181.977} C_DIS
LIN {X -10.6641,Y -137.2768,Z 178,A -91.0339,B 6.1678,C 0.4009,E1 6.1695,E2 183.2671} C_DIS
LIN {X -13.5262,Y -137.0234,Z 178,A -92.2645,B 6.1678,C 0.4012,E1 6.166,E2 184.5026} C_DIS
LIN {X -16.9565,Y -136.6423,Z 178,A -93.687,B 6.1678,C 0.4007,E1 6.1621,E2 185.9239} C_DIS
LIN {X -20.272,Y -136.1906,Z 178,A -95.08,B 6.1678,C 0.4004,E1 6.1582,E2 187.3176} C_DIS
LIN {X -23.4576,Y -135.6782,Z 178,A -96.4293,B 6.1679,C 0.4,E1 6.1545,E2 188.6682} C_DIS
LIN {X -26.1273,Y -135.1874,Z 178,A -97.603,B 6.1679,C 0.4,E1 6.1513,E2 189.8478} C_DIS
LIN {X -29.7133,Y -134.4461,Z 178,A -99.0969,B 6.1679,C 0.399,E1 6.1472,E2 191.3383} C_DIS
LIN {X -33.0685,Y -133.6612,Z 178,A -100.5391,B 6.168,C 0.3983,E1 6.1433,E2 192.782} C_DIS
LIN {X -35.7187,Y -132.9751,Z 178,A -101.7077,B 6.168,C 0.398,E1 6.1401,E2 193.9547} C_DIS
LIN {X -39.4924,Y -131.906,Z 178,A -103.3293,B 6.1681,C 0.3967,E1 6.1358,E2 195.5753} C_DIS
LIN {X -42.7003,Y -130.9027,Z 178,A -104.7388,B 6.1681,C 0.3958,E1 6.132,E2 196.9865} C_DIS
LIN {X -45.7564,Y -129.8652,Z 178,A -106.0926,B 6.1682,C 0.3949,E1 6.1284,E2 198.342} C_DIS
LIN {X -48.948,Y -128.6961,Z 178,A -107.519,B 6.1683,C 0.3938,E1 6.1247,E2 199.7701} C_DIS
LIN {X -52.1265,Y -127.4419,Z 178,A -108.954,B 6.1683,C 0.3926,E1 6.121,E2 201.207} C_DIS
LIN {X -55.2886,Y -126.1022,Z 178,A -110.3813,B 6.1685,C 0.3911,E1 6.1173,E2 202.6343} C_DIS
LIN {X -58.0991,Y -124.8307,Z 178,A -111.7276,B 6.1685,C 0.3905,E1 6.1139,E2 203.9887} C_DIS
LIN {X -61.5503,Y -123.1672,Z 178,A -113.3094,B 6.1686,C 0.3885,E1 6.1099,E2 205.569} C_DIS
LIN {X -65.3102,Y -121.2157,Z 178,A -115.1229,B 6.1687,C 0.3869,E1 6.1054,E2 207.389} C_DIS
LIN {X -69.0449,Y -119.1279,Z 178,A -116.9405,B 6.1689,C 0.3851,E1 6.101,E2 209.2115} C_DIS
LIN {X -72.3058,Y -117.1778,Z 178,A -118.4887,B 6.169,C 0.3825,E1 6.0973,E2 210.7555} C_DIS
LIN {X -75.6352,Y -115.0564,Z 178,A -120.2378,B 6.169,C 0.3814,E1 6.0931,E2 212.5181} C_DIS
LIN {X -78.9364,Y -112.8176,Z 178,A -121.8429,B 6.1693,C 0.3782,E1 6.0895,E2 214.116} C_DIS
LIN {X -81.8762,Y -110.7029,Z 178,A -123.459,B 6.1693,C 0.3771,E1 6.0858,E2 215.746} C_DIS
LIN {X -85.3425,Y -108.053,Z 178,A -125.2979,B 6.1695,C 0.3743,E1 6.0817,E2 217.5876} C_DIS
LIN {X -88.7792,Y -105.2475,Z 178,A -127.0859,B 6.1697,C 0.3704,E1 6.0779,E2 219.368} C_DIS
LIN {X -91.8459,Y -102.5815,Z 178,A -128.8655,B 6.1699,C 0.3684,E1 6.0742,E2 221.1585} C_DIS
LIN {X -94.8096,Y -99.8498,Z 178,A -130.4982,B 6.1701,C 0.3647,E1 6.0708,E2 222.7852} C_DIS
LIN {X -97.305,Y -97.4193,Z 178,A -132.0295,B 6.1701,C 0.3629,E1 6.0678,E2 224.3267} C_DIS
LIN {X -100.4058,Y -94.2203,Z 178,A -133.8562,B 6.1704,C 0.3589,E1 6.0643,E2 226.1494} C_DIS
LIN {X -102.8098,Y -91.591,Z 178,A -135.3725,B 6.1706,C 0.3562,E1 6.0614,E2 227.6696} C_DIS
LIN {X -105.5542,Y -88.4136,Z 178,A -137.1877,B 6.1707,C 0.3533,E1 6.0581,E2 229.4929} C_DIS
LIN {X -107.9578,Y -85.4628,Z 178,A -138.7626,B 6.1709,C 0.3497,E1 6.0553,E2 231.0662} C_DIS
LIN {X -110.2784,Y -82.4463,Z 178,A -140.4806,B 6.1711,C 0.3477,E1 6.0524,E2 232.8007} C_DIS
LIN {X -113.0105,Y -78.6592,Z 178,A -142.4074,B 6.1713,C 0.3431,E1 6.0493,E2 234.7247} C_DIS
LIN {X -115.2468,Y -75.3459,Z 178,A -144.0415,B 6.1716,C 0.3389,E1 6.0468,E2 236.3543} C_DIS
LIN {X -117.3854,Y -71.9675,Z 178,A -145.7964,B 6.1717,C 0.336,E1 6.0442,E2 238.12} C_DIS
LIN {X -119.6684,Y -68.1039,Z 178,A -147.6823,B 6.1719,C 0.3316,E1 6.0415,E2 240.0074} C_DIS
LIN {X -121.4615,Y -64.8528,Z 178,A -149.2242,B 6.1721,C 0.3278,E1 6.0395,E2 241.5482} C_DIS
LIN {X -122.9492,Y -61.9829,Z 178,A -150.5982,B 6.1723,C 0.3247,E1 6.0377,E2 242.9252} C_DIS
LIN {X -124.6115,Y -58.5732,Z 178,A -152.201,B 6.1725,C 0.321,E1 6.0358,E2 244.5302} C_DIS
LIN {X -125.8161,Y -55.9331,Z 178,A -153.4435,B 6.1726,C 0.3183,E1 6.0344,E2 245.7765} C_DIS
LIN {X -127.3838,Y -52.2704,Z 178,A -155.1261,B 6.1729,C 0.3142,E1 6.0325,E2 247.4614} C_DIS
LIN {X -128.642,Y -49.0926,Z 178,A -156.5783,B 6.173,C 0.3108,E1 6.0311,E2 248.9165} C_DIS
LIN {X -129.6907,Y -46.2458,Z 178,A -157.8922,B 6.1732,C 0.308,E1 6.0298,E2 250.2361} C_DIS
LIN {X -130.7451,Y -43.1738,Z 178,A -159.263,B 6.1733,C 0.3045,E1 6.0286,E2 251.6084} C_DIS
LIN {X -131.8615,Y -39.6379,Z 178,A -160.8242,B 6.1735,C 0.3006,E1 6.0273,E2 253.171} C_DIS
LIN {X -132.7845,Y -36.4264,Z 178,A -162.2452,B 6.1737,C 0.2971,E1 6.0262,E2 254.595} C_DIS
LIN {X -133.6242,Y -33.2142,Z 178,A -163.6561,B 6.1739,C 0.2936,E1 6.0252,E2 256.0087} C_DIS
LIN {X -134.3804,Y -30.0089,Z 178,A -165.0598,B 6.174,C 0.2901,E1 6.0244,E2 257.4156} C_DIS
LIN {X -135.0866,Y -26.6541,Z 178,A -166.5157,B 6.1742,C 0.2865,E1 6.0236,E2 258.8743} C_DIS
LIN {X -135.6156,Y -23.8077,Z 178,A -167.7422,B 6.1743,C 0.2833,E1 6.0229,E2 260.1026} C_DIS
LIN {X -136.1254,Y -20.6932,Z 178,A -169.1126,B 6.1745,C 0.2802,E1 6.0223,E2 261.4792} C_DIS
LIN {X -136.6064,Y -17.2435,Z 178,A -170.5751,B 6.1747,C 0.2763,E1 6.0218,E2 262.9424} C_DIS
LIN {X -136.9833,Y -13.9435,Z 178,A -171.9831,B 6.1748,C 0.2726,E1 6.0214,E2 264.3526} C_DIS
LIN {X -137.2073,Y -11.5065,Z 178,A -173.0632,B 6.1749,C 0.2704,E1 6.0211,E2 265.4396} C_DIS
LIN {X -137.4535,Y -8.0581,Z 178,A -174.5215,B 6.1751,C 0.2665,E1 6.0208,E2 266.8993} C_DIS
LIN {X -137.6145,Y -4.5941,Z 178,A -175.97,B 6.1753,C 0.2624,E1 6.0207,E2 268.3474} C_DIS
LIN {X -137.6827,Y -1.5247,Z 178,A -177.2722,B 6.1754,C 0.259,E1 6.0207,E2 269.6516} C_DIS
LIN {X -137.6752,Y 1.9764,Z 178,A -178.8299,B 6.1755,C 0.2559,E1 6.0207,E2 271.2208} C_DIS
LIN {X -137.578,Y 5.5277,Z 178,A 179.6579,B 6.1757,C 0.252,E1 6.0207,E2 272.736} C_DIS
LIN {X -137.3804,Y 9.2443,Z 178,A 178.1236,B 6.1759,C 0.2474,E1 6.0211,E2 274.2673} C_DIS
LIN {X -137.1341,Y 12.3722,Z 178,A 176.7836,B 6.176,C 0.2441,E1 6.0214,E2 275.6105} C_DIS
LIN {X -136.8774,Y 14.9271,Z 178,A 175.657,B 6.1761,C 0.2416,E1 6.0217,E2 276.7433} C_DIS
LIN {X -136.4929,Y 18.1094,Z 178,A 174.2975,B 6.1762,C 0.2381,E1 6.0222,E2 278.105} C_DIS
LIN {X -135.9442,Y 21.8633,Z 178,A 172.6998,B 6.1764,C 0.2338,E1 6.0229,E2 279.7037} C_DIS
LIN {X -135.3924,Y 25.0547,Z 178,A 171.3179,B 6.1765,C 0.2304,E1 6.0235,E2 281.0887} C_DIS
LIN {X -134.7903,Y 28.1103,Z 178,A 170.0037,B 6.1767,C 0.2269,E1 6.0243,E2 282.404} C_DIS
LIN {X -134.0814,Y 31.3176,Z 178,A 168.5822,B 6.1767,C 0.2237,E1 6.0251,E2 283.8312} C_DIS
LIN {X -133.2536,Y 34.6745,Z 178,A 167.1124,B 6.1769,C 0.22,E1 6.0261,E2 285.3035} C_DIS
LIN {X -132.3761,Y 37.8868,Z 178,A 165.6919,B 6.177,C 0.2166,E1 6.0272,E2 286.7271} C_DIS
LIN {X -131.4971,Y 40.8284,Z 178,A 164.3678,B 6.1771,C 0.2135,E1 6.0283,E2 288.0559} C_DIS
LIN {X -130.4178,Y 44.1567,Z 178,A 162.8916,B 6.1773,C 0.2098,E1 6.0296,E2 289.5333} C_DIS
LIN {X -129.2913,Y 47.3536,Z 178,A 161.4467,B 6.1773,C 0.2063,E1 6.031,E2 290.9812} C_DIS
LIN {X -128.0797,Y 50.5391,Z 178,A 159.9948,B 6.1775,C 0.2029,E1 6.0324,E2 292.4359} C_DIS
LIN {X -126.8592,Y 53.5267,Z 178,A 158.6332,B 6.1776,C 0.1995,E1 6.0339,E2 293.7986} C_DIS
LIN {X -125.48,Y 56.6845,Z 178,A 157.1393,B 6.1777,C 0.1964,E1 6.0356,E2 295.2986} C_DIS
LIN {X -123.9328,Y 59.9938,Z 178,A 155.5981,B 6.1778,C 0.1927,E1 6.0374,E2 296.8411} C_DIS
LIN {X -122.3088,Y 63.2408,Z 178,A 154.0535,B 6.1779,C 0.1892,E1 6.0394,E2 298.3885} C_DIS
LIN {X -120.7038,Y 66.2523,Z 178,A 152.5174,B 6.178,C 0.1868,E1 6.0415,E2 299.9376} C_DIS
LIN {X -118.5397,Y 70.0508,Z 178,A 150.7429,B 6.1781,C 0.1819,E1 6.0439,E2 301.705} C_DIS
LIN {X -116.7136,Y 73.0528,Z 178,A 149.2497,B 6.1782,C 0.1786,E1 6.0461,E2 303.2007} C_DIS
LIN {X -114.8058,Y 76.0158,Z 178,A 147.7441,B 6.1783,C 0.1755,E1 6.0484,E2 304.7097} C_DIS
LIN {X -112.4699,Y 79.4303,Z 178,A 145.9446,B 6.1784,C 0.1723,E1 6.0513,E2 306.5174} C_DIS
LIN {X -110.1735,Y 82.5872,Z 178,A 144.2932,B 6.1785,C 0.1689,E1 6.054,E2 308.1706} C_DIS
LIN {X -107.5616,Y 85.9605,Z 178,A 142.445,B 6.1786,C 0.1657,E1 6.0572,E2 310.0261} C_DIS
LIN {X -104.6716,Y 89.4574,Z 178,A 140.6063,B 6.1787,C 0.161,E1 6.0605,E2 311.8571} C_DIS
LIN {X -102.2696,Y 92.1942,Z 178,A 138.9427,B 6.1787,C 0.1594,E1 6.0637,E2 313.5376} C_DIS
LIN {X -99.2342,Y 95.4537,Z 178,A 137.086,B 6.1789,C 0.1556,E1 6.0672,E2 315.3931} C_DIS
LIN {X -96.0939,Y 98.6144,Z 178,A 135.2999,B 6.1789,C 0.1511,E1 6.0707,E2 317.1692} C_DIS
LIN {X -93.5687,Y 101.0133,Z 178,A 133.8186,B 6.179,C 0.1486,E1 6.0738,E2 318.6532} C_DIS
LIN {X -90.6125,Y 103.6727,Z 178,A 132.0481,B 6.179,C 0.1468,E1 6.0775,E2 320.4364} C_DIS
LIN {X -87.2723,Y 106.4998,Z 178,A 130.1946,B 6.1791,C 0.1438,E1 6.0815,E2 322.2923} C_DIS
LIN {X -83.9999,Y 109.1002,Z 178,A 128.525,B 6.1792,C 0.14,E1 6.0851,E2 323.952} C_DIS
LIN {X -81.2269,Y 111.1799,Z 178,A 126.9807,B 6.1792,C 0.1387,E1 6.0886,E2 325.5075} C_DIS
LIN {X -77.5479,Y 113.7768,Z 178,A 125.1721,B 6.1793,C 0.1349,E1 6.0927,E2 327.3067} C_DIS
LIN {X -74.5394,Y 115.7699,Z 178,A 123.5261,B 6.1793,C 0.1342,E1 6.0966,E2 328.9691} C_DIS
LIN {X -70.7064,Y 118.1495,Z 178,A 121.6321,B 6.1794,C 0.1317,E1 6.1011,E2 330.8636} C_DIS
LIN {X -66.8387,Y 120.3796,Z 178,A 119.778,B 6.1794,C 0.129,E1 6.1056,E2 332.7158} C_DIS
LIN {X -63.3806,Y 122.2354,Z 178,A 118.2163,B 6.1795,C 0.126,E1 6.1095,E2 334.2675} C_DIS
LIN {X -60.4803,Y 123.695,Z 178,A 116.8389,B 6.1795,C 0.1246,E1 6.1129,E2 335.6471} C_DIS
LIN {X -57.4211,Y 125.1442,Z 178,A 115.4056,B 6.1795,C 0.1233,E1 6.1166,E2 337.0824} C_DIS
LIN {X -53.8534,Y 126.7228,Z 178,A 113.7939,B 6.1796,C 0.1213,E1 6.1207,E2 338.6916} C_DIS
LIN {X -50.6834,Y 128.0236,Z 178,A 112.357,B 6.1796,C 0.1199,E1 6.1244,E2 340.1288} C_DIS
LIN {X -47.4985,Y 129.2391,Z 178,A 110.9286,B 6.1796,C 0.1187,E1 6.1281,E2 341.5575} C_DIS
LIN {X -44.3019,Y 130.3694,Z 178,A 109.5089,B 6.1797,C 0.1175,E1 6.1319,E2 342.9773} C_DIS
LIN {X -41.3363,Y 131.3385,Z 178,A 108.1979,B 6.1797,C 0.1165,E1 6.1354,E2 344.2889} C_DIS
LIN {X -38.0324,Y 132.3335,Z 178,A 106.7597,B 6.1797,C 0.1154,E1 6.1392,E2 345.7265} C_DIS
LIN {X -34.8202,Y 133.2147,Z 178,A 105.3844,B 6.1797,C 0.1143,E1 6.1429,E2 347.0996} C_DIS
LIN {X -31.9706,Y 133.9259,Z 178,A 104.0941,B 6.1797,C 0.1143,E1 6.1465,E2 348.3974} C_DIS
LIN {X -28.2556,Y 134.7608,Z 178,A 102.5506,B 6.1797,C 0.1129,E1 6.1507,E2 349.9351} C_DIS
LIN {X -25.0547,Y 135.3924,Z 178,A 101.1896,B 6.1797,C 0.1123,E1 6.1544,E2 351.2957} C_DIS
LIN {X -22.0079,Y 135.9201,Z 178,A 99.8998,B 6.1798,C 0.1117,E1 6.1579,E2 352.5851} C_DIS
LIN {X -19.2104,Y 136.3423,Z 178,A 98.683,B 6.1798,C 0.1117,E1 6.1613,E2 353.806} C_DIS
LIN {X -15.5195,Y 136.8137,Z 178,A 97.171,B 6.1798,C 0.1108,E1 6.1655,E2 355.3128} C_DIS
LIN {X -12.5147,Y 137.1205,Z 178,A 95.9301,B 6.1798,C 0.1103,E1 6.1689,E2 356.5511} C_DIS
LIN {X -9.2443,Y 137.3804,Z 178,A 94.5491,B 6.1798,C 0.1103,E1 6.1728,E2 357.9334} C_DIS
LIN {X -6.1383,Y 137.5542,Z 178,A 93.256,B 6.1798,C 0.1101,E1 6.1764,E2 359.2258} C_DIS
LIN {X -3.5953,Y 137.6422,Z 178,A 92.147,B 6.1798,C 0.1106,E1 6.1795,E2 360.3403} C_DIS
LIN {X 0,Y 137.6911,Z 178,A 90.7041,B 6.1798,C 0.1099,E1 6.1835,E2 361.776} C_DIS
LIN {X 2.9173,Y 137.6595,Z 178,A 89.4837,B 6.1798,C 0.1101,E1 6.1869,E2 362.9967} C_DIS
LIN {X 5.9983,Y 137.5597,Z 178,A 88.2041,B 6.1798,C 0.1102,E1 6.1905,E2 364.2754} C_DIS
LIN {X 9.2443,Y 137.3804,Z 178,A 86.8512,B 6.1798,C 0.1105,E1 6.1943,E2 365.6278} C_DIS
LIN {X 12.3722,Y 137.1341,Z 178,A 85.5457,B 6.1798,C 0.1109,E1 6.1979,E2 366.9328} C_DIS
LIN {X 15.3766,Y 136.8291,Z 178,A 84.2903,B 6.1798,C 0.1112,E1 6.2014,E2 368.1875} C_DIS
LIN {X 18.684,Y 136.4175,Z 178,A 82.9055,B 6.1798,C 0.1118,E1 6.2052,E2 369.5717} C_DIS
LIN {X 22.7534,Y 135.7957,Z 178,A 81.1742,B 6.1798,C 0.1128,E1 6.21,E2 371.3046} C_DIS
LIN {X 26.5091,Y 135.1144,Z 178,A 79.6122,B 6.1798,C 0.1133,E1 6.2143,E2 372.8629} C_DIS
LIN {X 29.7133,Y 134.4461,Z 178,A 78.2548,B 6.1798,C 0.1141,E1 6.218,E2 374.2194} C_DIS
LIN {X 32.7978,Y 133.7265,Z 178,A 76.958,B 6.1798,C 0.1147,E1 6.2215,E2 375.5133} C_DIS
LIN {X 36.2808,Y 132.8253,Z 178,A 75.4528,B 6.1798,C 0.116,E1 6.2256,E2 377.0192} C_DIS
LIN {X 39.4924,Y 131.906,Z 178,A 74.0701,B 6.1798,C 0.117,E1 6.2293,E2 378.4007} C_DIS
LIN {X 42.4059,Y 130.9968,Z 178,A 72.7975,B 6.1797,C 0.1182,E1 6.2327,E2 379.6733} C_DIS
LIN {X 45.4725,Y 129.9636,Z 178,A 71.4785,B 6.1797,C 0.119,E1 6.2361,E2 380.9887} C_DIS
LIN {X 48.948,Y 128.6961,Z 178,A 69.9413,B 6.1797,C 0.1206,E1 6.2402,E2 382.5254} C_DIS
LIN {X 52.1265,Y 127.4419,Z 178,A 68.5302,B 6.1797,C 0.122,E1 6.2438,E2 383.935} C_DIS
LIN {X 54.9976,Y 126.228,Z 178,A 67.2062,B 6.1796,C 0.1238,E1 6.2472,E2 385.2621} C_DIS
LIN {X 58.431,Y 124.6772,Z 178,A 65.69,B 6.1796,C 0.125,E1 6.251,E2 386.7719} C_DIS
LIN {X 61.5466,Y 123.169,Z 178,A 64.2583,B 6.1796,C 0.1267,E1 6.2546,E2 388.2025} C_DIS
LIN {X 64.9596,Y 121.4041,Z 178,A 62.5777,B 6.1795,C 0.13,E1 6.2588,E2 389.8932} C_DIS
LIN {X 68.6051,Y 119.3825,Z 178,A 60.9725,B 6.1795,C 0.1306,E1 6.2627,E2 391.4825} C_DIS
LIN {X 71.5565,Y 117.6369,Z 178,A 59.4984,B 6.1794,C 0.1334,E1 6.2662,E2 392.9623} C_DIS
LIN {X 75.2789,Y 115.2904,Z 178,A 57.7368,B 6.1794,C 0.1352,E1 6.2703,E2 394.7155} C_DIS
LIN {X 78.2104,Y 113.3222,Z 178,A 56.2859,B 6.1793,C 0.1373,E1 6.2737,E2 396.1643} C_DIS
LIN {X 81.1622,Y 111.2274,Z 178,A 54.6959,B 6.1793,C 0.1411,E1 6.2773,E2 397.7647} C_DIS
LIN {X 84.7346,Y 108.5304,Z 178,A 52.8534,B 6.1791,C 0.1441,E1 6.2814,E2 399.605} C_DIS
LIN {X 88.1589,Y 105.7679,Z 178,A 51.1198,B 6.1791,C 0.1459,E1 6.2851,E2 401.3269} C_DIS
LIN {X 91.4704,Y 102.9172,Z 178,A 49.3678,B 6.1791,C 0.1483,E1 6.2888,E2 403.0711} C_DIS
LIN {X 94.1615,Y 100.4612,Z 178,A 47.8835,B 6.179,C 0.1508,E1 6.2918,E2 404.5518} C_DIS
LIN {X 96.6725,Y 98.047,Z 178,A 46.3947,B 6.1789,C 0.1543,E1 6.2948,E2 406.0458} C_DIS
LIN {X 99.794,Y 94.868,Z 178,A 44.6345,B 6.1789,C 0.1566,E1 6.2982,E2 407.7948} C_DIS
LIN {X 102.2153,Y 92.254,Z 178,A 43.0892,B 6.1787,C 0.1607,E1 6.3011,E2 409.3482} C_DIS
LIN {X 105.1956,Y 88.841,Z 178,A 41.3329,B 6.1787,C 0.1628,E1 6.3043,E2 411.0891} C_DIS
LIN {X 107.4548,Y 86.0948,Z 178,A 39.8802,B 6.1787,C 0.1656,E1 6.3069,E2 412.539} C_DIS
LIN {X 109.6392,Y 83.2951,Z 178,A 38.3201,B 6.1785,C 0.1703,E1 6.3095,E2 414.1099} C_DIS
LIN {X 112.2153,Y 79.7904,Z 178,A 36.639,B 6.1785,C 0.1724,E1 6.3123,E2 415.7755} C_DIS
LIN {X 114.2269,Y 76.8829,Z 178,A 35.2102,B 6.1783,C 0.1752,E1 6.3145,E2 417.1997} C_DIS
LIN {X 116.3637,Y 73.6082,Z 178,A 33.5193,B 6.1782,C 0.1801,E1 6.3171,E2 418.8991} C_DIS
LIN {X 118.4587,Y 70.1877,Z 178,A 31.9668,B 6.1782,C 0.1823,E1 6.3193,E2 420.4379} C_DIS
LIN {X 120.2448,Y 67.0823,Z 178,A 30.5152,B 6.178,C 0.1854,E1 6.3213,E2 421.8853} C_DIS
LIN {X 122.0997,Y 63.639,Z 178,A 28.8989,B 6.178,C 0.1893,E1 6.3234,E2 423.5009} C_DIS
LIN {X 123.8651,Y 60.1354,Z 178,A 27.3247,B 6.1778,C 0.1926,E1 6.3253,E2 425.0688} C_DIS
LIN {X 125.1301,Y 57.4516,Z 178,A 26.0883,B 6.1778,C 0.1958,E1 6.3268,E2 426.306} C_DIS
LIN {X 126.7228,Y 53.8534,Z 178,A 24.5157,B 6.1776,C 0.199,E1 6.3285,E2 427.8714} C_DIS
LIN {X 128.0236,Y 50.6834,Z 178,A 23.1217,B 6.1776,C 0.2023,E1 6.33,E2 429.2623} C_DIS
LIN {X 129.2391,Y 47.4985,Z 178,A 21.7355,B 6.1774,C 0.2055,E1 6.3314,E2 430.6453} C_DIS
LIN {X 130.2288,Y 44.7075,Z 178,A 20.5385,B 6.1774,C 0.2082,E1 6.3324,E2 431.8385} C_DIS
LIN {X 131.2362,Y 41.6566,Z 178,A 19.2087,B 6.1772,C 0.2117,E1 6.3336,E2 433.1682} C_DIS
LIN {X 132.2653,Y 38.2652,Z 178,A 17.7816,B 6.1771,C 0.215,E1 6.3347,E2 434.5902} C_DIS
LIN {X 133.1087,Y 35.218,Z 178,A 16.4605,B 6.177,C 0.2187,E1 6.3357,E2 435.9129} C_DIS
LIN {X 134.0131,Y 31.6087,Z 178,A 14.9847,B 6.1768,C 0.2218,E1 6.3367,E2 437.3806} C_DIS
LIN {X 134.7608,Y 28.2556,Z 178,A 13.5935,B 6.1768,C 0.2252,E1 6.3375,E2 438.768} C_DIS
LIN {X 135.2912,Y 25.5843,Z 178,A 12.4504,B 6.1766,C 0.2285,E1 6.3381,E2 439.913} C_DIS
LIN {X 135.9201,Y 22.0079,Z 178,A 11.0131,B 6.1765,C 0.2315,E1 6.3388,E2 441.3422} C_DIS
LIN {X 136.397,Y 18.8281,Z 178,A 9.7081,B 6.1764,C 0.2348,E1 6.3393,E2 442.644} C_DIS
LIN {X 136.8137,Y 15.5195,Z 178,A 8.3542,B 6.1762,C 0.2381,E1 6.3397,E2 443.9947} C_DIS
LIN {X 137.1205,Y 12.5147,Z 178,A 7.1493,B 6.1762,C 0.2408,E1 6.34,E2 445.1939} C_DIS
LIN {X 137.3804,Y 9.2443,Z 178,A 5.7969,B 6.176,C 0.2445,E1 6.3403,E2 446.5458} C_DIS
LIN {X 137.5542,Y 6.1383,Z 178,A 4.5347,B 6.1759,C 0.2477,E1 6.3405,E2 447.8049} C_DIS
LIN {X 137.6533,Y 3.1957,Z 178,A 3.3356,B 6.1757,C 0.2507,E1 6.3405,E2 449.0016} C_DIS
LIN {X 137.6912,Y 0,Z 178,A 2.0584,B 6.1757,C 0.2537,E1 6.3406,E2 450.2732} C_DIS
LIN {X 137.6572,Y -3.0562,Z 178,A 0.7968,B 6.1755,C 0.2571,E1 6.3406,E2 451.5345} C_DIS
LIN {X 137.5597,Y -5.9983,Z 178,A -0.4025,B 6.1754,C 0.2602,E1 6.3404,E2 452.7315} C_DIS
LIN {X 137.3804,Y -9.2443,Z 178,A -1.7264,B 6.1752,C 0.2636,E1 6.3402,E2 454.0529} C_DIS
LIN {X 137.1341,Y -12.3722,Z 178,A -3.0047,B 6.1751,C 0.2669,E1 6.3399,E2 455.3288} C_DIS
LIN {X 136.8291,Y -15.3766,Z 178,A -4.2165,B 6.175,C 0.2697,E1 6.3396,E2 456.536} C_DIS
LIN {X 136.4175,Y -18.684,Z 178,A -5.5921,B 6.1748,C 0.2734,E1 6.3391,E2 457.9114} C_DIS
LIN {X 135.9981,Y -21.5153,Z 178,A -6.7752,B 6.1746,C 0.2767,E1 6.3386,E2 459.0944} C_DIS
LIN {X 135.3924,Y -25.0547,Z 178,A -8.2202,B 6.1745,C 0.2801,E1 6.3379,E2 460.5345} C_DIS
LIN {X 134.8276,Y -27.927,Z 178,A -9.3956,B 6.1744,C 0.2828,E1 6.3372,E2 461.7054} C_DIS
LIN {X 134.0814,Y -31.3176,Z 178,A -10.8319,B 6.1742,C 0.2867,E1 6.3363,E2 463.142} C_DIS
LIN {X 133.2536,Y -34.6745,Z 178,A -12.2356,B 6.174,C 0.2901,E1 6.3354,E2 464.5426} C_DIS
LIN {X 132.3761,Y -37.8868,Z 178,A -13.5927,B 6.1739,C 0.2935,E1 6.3343,E2 465.8972} C_DIS
LIN {X 131.4149,Y -41.097,Z 178,A -14.9576,B 6.1737,C 0.2969,E1 6.3332,E2 467.2596} C_DIS
LIN {X 130.4178,Y -44.1567,Z 178,A -16.2691,B 6.1736,C 0.3001,E1 6.3321,E2 468.5688} C_DIS
LIN {X 129.2913,Y -47.3536,Z 178,A -17.6508,B 6.1734,C 0.3034,E1 6.3308,E2 469.9481} C_DIS
LIN {X 128.0797,Y -50.5391,Z 178,A -19.0397,B 6.1732,C 0.3068,E1 6.3294,E2 471.3345} C_DIS
LIN {X 126.7827,Y -53.7098,Z 178,A -20.4361,B 6.1731,C 0.3101,E1 6.3279,E2 472.7285} C_DIS
LIN {X 125.3731,Y -56.9234,Z 178,A -21.8653,B 6.1729,C 0.3134,E1 6.3263,E2 474.1551} C_DIS
LIN {X 123.9328,Y -59.9938,Z 178,A -23.2494,B 6.1727,C 0.3167,E1 6.3246,E2 475.5371} C_DIS
LIN {X 122.3088,Y -63.2408,Z 178,A -24.7298,B 6.1726,C 0.3201,E1 6.3227,E2 477.015} C_DIS
LIN {X 121.0861,Y -65.5514,Z 178,A -25.8978,B 6.1723,C 0.3242,E1 6.3212,E2 478.1942} C_DIS
LIN {X 118.9834,Y -69.2945,Z 178,A -27.5558,B 6.1723,C 0.3266,E1 6.3189,E2 479.8374} C_DIS
LIN {X 116.8679,Y -72.8049,Z 178,A -29.2714,B 6.172,C 0.331,E1 6.3164,E2 481.5559} C_DIS
LIN {X 114.4467,Y -76.5547,Z 178,A -31.0742,B 6.1718,C 0.3346,E1 6.3136,E2 483.3534} C_DIS
LIN {X 112.2619,Y -79.7251,Z 178,A -32.6138,B 6.1716,C 0.3374,E1 6.3112,E2 484.8865} C_DIS
LIN {X 110.1735,Y -82.5872,Z 178,A -34.061,B 6.1715,C 0.3405,E1 6.3088,E2 486.3315} C_DIS
LIN {X 108.008,Y -85.3998,Z 178,A -35.5602,B 6.1713,C 0.3442,E1 6.3062,E2 487.8349} C_DIS
LIN {X 105.2475,Y -88.7792,Z 178,A -37.2941,B 6.1711,C 0.347,E1 6.3031,E2 489.56} C_DIS
LIN {X 102.9172,Y -91.4704,Z 178,A -38.7573,B 6.1709,C 0.35,E1 6.3004,E2 491.0222} C_DIS
LIN {X 100.4612,Y -94.1615,Z 178,A -40.256,B 6.1708,C 0.353,E1 6.2976,E2 492.52} C_DIS
LIN {X 97.5484,Y -97.175,Z 178,A -41.9865,B 6.1706,C 0.3565,E1 6.2942,E2 494.2503} C_DIS
LIN {X 94.868,Y -99.794,Z 178,A -43.4866,B 6.1704,C 0.3587,E1 6.2912,E2 495.7442} C_DIS
LIN {X 92.254,Y -102.2153,Z 178,A -44.9533,B 6.1703,C 0.3614,E1 6.2882,E2 497.2102} C_DIS
LIN {X 89.5189,Y -104.6194,Z 178,A -46.5105,B 6.1701,C 0.3651,E1 6.2849,E2 498.7741} C_DIS
LIN {X 86.0948,Y -107.4548,Z 178,A -48.2495,B 6.17,C 0.3668,E1 6.2812,E2 500.5004} C_DIS
LIN {X 83.359,Y -109.5904,Z 178,A -49.6794,B 6.1698,C 0.3692,E1 6.278,E2 501.9297} C_DIS
LIN {X 80.5102,Y -111.7,Z 178,A -51.1328,B 6.1697,C 0.3715,E1 6.2747,E2 503.3815} C_DIS
LIN {X 77.3364,Y -113.92,Z 178,A -52.8142,B 6.1695,C 0.3754,E1 6.2708,E2 505.0733} C_DIS
LIN {X 73.6407,Y -116.3432,Z 178,A -54.6337,B 6.1693,C 0.3781,E1 6.2666,E2 506.8918} C_DIS
LIN {X 70.1877,Y -118.4587,Z 178,A -56.2052,B 6.1693,C 0.3789,E1 6.2628,E2 508.45} C_DIS
LIN {X 67.0823,Y -120.2448,Z 178,A -57.6935,B 6.1691,C 0.3812,E1 6.2592,E2 509.9393} C_DIS
LIN {X 63.3806,Y -122.2354,Z 178,A -59.3953,B 6.169,C 0.3829,E1 6.255,E2 511.6363} C_DIS
LIN {X 60.1354,Y -123.8651,Z 178,A -60.8883,B 6.1689,C 0.3847,E1 6.2513,E2 513.1281} C_DIS
LIN {X 57.0052,Y -125.3366,Z 178,A -62.311,B 6.1688,C 0.3864,E1 6.2477,E2 514.5498} C_DIS
LIN {X 54.2079,Y -126.5695,Z 178,A -63.5944,B 6.1687,C 0.3881,E1 6.2444,E2 515.8356} C_DIS
LIN {X 50.6834,Y -128.0236,Z 178,A -65.1385,B 6.1686,C 0.3894,E1 6.2404,E2 517.3754} C_DIS
LIN {X 47.4985,Y -129.2391,Z 178,A -66.5424,B 6.1686,C 0.3907,E1 6.2367,E2 518.7784} C_DIS
LIN {X 44.3019,Y -130.3694,Z 178,A -67.9392,B 6.1684,C 0.392,E1 6.2331,E2 520.1744} C_DIS
LIN {X 41.2424,Y -131.3685,Z 178,A -69.2661,B 6.1684,C 0.3931,E1 6.2295,E2 521.5005} C_DIS
LIN {X 38.0324,Y -132.3335,Z 178,A -70.6486,B 6.1683,C 0.3942,E1 6.2258,E2 522.8824} C_DIS
LIN {X 34.8202,Y -133.2147,Z 178,A -72.0228,B 6.1683,C 0.3952,E1 6.2221,E2 524.2561} C_DIS
LIN {X 31.9892,Y -133.9214,Z 178,A -73.2184,B 6.1682,C 0.3959,E1 6.2189,E2 525.4499} C_DIS
LIN {X 28.6442,Y -134.6769,Z 178,A -74.6719,B 6.1681,C 0.3973,E1 6.2149,E2 526.9078} C_DIS
LIN {X 25.0547,Y -135.3924,Z 178,A -76.1559,B 6.1681,C 0.3978,E1 6.2109,E2 528.3878} C_DIS
LIN {X 22.0079,Y -135.9201,Z 178,A -77.4284,B 6.1681,C 0.3983,E1 6.2073,E2 529.6592} C_DIS
LIN {X 18.8281,Y -136.397,Z 178,A -78.7642,B 6.168,C 0.399,E1 6.2037,E2 530.9955} C_DIS
LIN {X 16.1711,Y -136.736,Z 178,A -79.9006,B 6.168,C 0.3998,E1 6.2005,E2 532.1353} C_DIS
LIN {X 12.5147,Y -137.1205,Z 178,A -81.3951,B 6.168,C 0.4,E1 6.1964,E2 533.6261} C_DIS
LIN {X 9.2443,Y -137.3804,Z 178,A -82.7539,B 6.1679,C 0.4003,E1 6.1926,E2 534.9848} C_DIS
LIN {X 6.1383,Y -137.5542,Z 178,A -84.043,B 6.1679,C 0.4006,E1 6.189,E2 536.2738} C_DIS
LIN {X 3.1957,Y -137.6533,Z 178,A -85.2476,B 6.1679,C 0.4006,E1 6.1856,E2 537.4764} C_DIS
LIN {X 3.1957,Y -137.6533,Z 178,A -85.2476,B 6.1679,C 0.4006,E1 6.1856,E2 537.4764} C_DIS
Enddeposition()
LIN {X 1.0123,Y -138.5881,Z 178,A -85.6322,B 6.1071,C 0.3963,E1 6.1237,E2 537.8431} C_DIS
Startdeposition()
$VEL.CP = VEL_PRINT
LIN {X 4.4203,Y -138.5239,Z 178,A -84.1718,B 6.1071,C 0.3954,E1 6.1278,E2 536.3754} C_DIS
LIN {X 7.0621,Y -138.4131,Z 178,A -83.0297,B 6.1072,C 0.3944,E1 6.131,E2 535.2262} C_DIS
LIN {X 10.9595,Y -138.1609,Z 178,A -81.4681,B 6.1072,C 0.3946,E1 6.1353,E2 533.6709} C_DIS
LIN {X 13.4325,Y -137.9407,Z 178,A -80.4024,B 6.1072,C 0.3936,E1 6.1383,E2 532.5993} C_DIS
LIN {X 17.2367,Y -137.5192,Z 178,A -78.0988,B 6.108,C 0.3824,E1 6.145,E2 530.1992} C_DIS
LIN {X 22.7176,Y -136.7184,Z 178,A -76.415,B 6.1075,C 0.39,E1 6.1494,E2 528.5946} C_DIS
LIN {X 27.3173,Y -135.8745,Z 178,A -74.5203,B 6.1075,C 0.3893,E1 6.1545,E2 526.7039} C_DIS
LIN {X 31.2584,Y -135.0225,Z 178,A -72.7239,B 6.1078,C 0.3861,E1 6.1595,E2 524.8893} C_DIS
LIN {X 36.4296,Y -133.7214,Z 178,A -70.7951,B 6.1076,C 0.3884,E1 6.1646,E2 522.9955} C_DIS
LIN {X 39.8936,Y -132.7288,Z 178,A -69.3451,B 6.1076,C 0.3876,E1 6.1685,E2 521.5497} C_DIS
LIN {X 42.3509,Y -131.9636,Z 178,A -68.2562,B 6.1078,C 0.3862,E1 6.1714,E2 520.4567} C_DIS
LIN {X 45.5329,Y -130.8997,Z 178,A -66.7873,B 6.1079,C 0.3835,E1 6.1753,E2 518.9761} C_DIS
LIN {X 48.9875,Y -129.6469,Z 178,A -65.3588,B 6.1079,C 0.3832,E1 6.179,E2 517.5584} C_DIS
LIN {X 52.1551,Y -128.4053,Z 178,A -63.9581,B 6.108,C 0.3817,E1 6.1827,E2 516.1575} C_DIS
LIN {X 55.226,Y -127.1144,Z 178,A -62.5851,B 6.1081,C 0.38,E1 6.1862,E2 514.784} C_DIS
LIN {X 58.5442,Y -125.6211,Z 178,A -61.1218,B 6.1082,C 0.3787,E1 6.1899,E2 513.3249} C_DIS
LIN {X 62.0489,Y -123.9295,Z 178,A -59.5116,B 6.1084,C 0.3765,E1 6.1939,E2 511.7134} C_DIS
LIN {X 64.9157,Y -122.4506,Z 178,A -58.179,B 6.1084,C 0.3746,E1 6.1972,E2 510.3799} C_DIS
LIN {X 69.2861,Y -120.0331,Z 178,A -56.0539,B 6.1087,C 0.3706,E1 6.2024,E2 508.2451} C_DIS
LIN {X 72.9504,Y -117.8423,Z 178,A -54.3323,B 6.1089,C 0.3685,E1 6.2065,E2 506.5279} C_DIS
LIN {X 76.5415,Y -115.5423,Z 178,A -52.6016,B 6.1089,C 0.3661,E1 6.2106,E2 504.8} C_DIS
LIN {X 81.44,Y -112.1428,Z 178,A -50.2319,B 6.1092,C 0.3633,E1 6.216,E2 502.4407} C_DIS
LIN {X 85.1385,Y -109.3617,Z 178,A -48.1851,B 6.1095,C 0.3577,E1 6.2205,E2 500.3746} C_DIS
LIN {X 88.9564,Y -106.2791,Z 178,A -45.4902,B 6.1103,C 0.343,E1 6.2265,E2 497.5896} C_DIS
LIN {X 93.9027,Y -101.9352,Z 178,A -43.9057,B 6.1096,C 0.3561,E1 6.2295,E2 496.1532} C_DIS
LIN {X 97.3467,Y -98.6523,Z 178,A -41.651,B 6.1101,C 0.3473,E1 6.2341,E2 493.859} C_DIS
LIN {X 101.9319,Y -93.9062,Z 178,A -38.9858,B 6.1104,C 0.3425,E1 6.2392,E2 491.1997} C_DIS
LIN {X 106.54,Y -88.6442,Z 178,A -36.3294,B 6.1104,C 0.34,E1 6.244,E2 488.5716} C_DIS
LIN {X 108.1984,Y -86.6123,Z 178,A -34.8521,B 6.111,C 0.331,E1 6.2467,E2 487.0416} C_DIS
LIN {X 110.3437,Y -83.8624,Z 178,A -33.7965,B 6.1108,C 0.334,E1 6.2484,E2 486.0355} C_DIS
LIN {X 112.1061,Y -81.4907,Z 178,A -32.5451,B 6.111,C 0.3307,E1 6.2505,E2 484.779} C_DIS
LIN {X 114.5086,Y -78.0796,Z 178,A -30.8271,B 6.1112,C 0.3266,E1 6.2532,E2 483.0604} C_DIS
LIN {X 116.8938,Y -74.4607,Z 178,A -28.874,B 6.1116,C 0.3196,E1 6.2562,E2 481.0844} C_DIS
LIN {X 119.5594,Y -70.1002,Z 178,A -26.9709,B 6.1116,C 0.3178,E1 6.2589,E2 479.2069} C_DIS
LIN {X 121.807,Y -66.1181,Z 178,A -25.085,B 6.1119,C 0.313,E1 6.2614,E2 477.3198} C_DIS
LIN {X 123.6021,Y -62.6935,Z 178,A -23.5565,B 6.1121,C 0.3101,E1 6.2634,E2 475.7989} C_DIS
LIN {X 125.8333,Y -58.0854,Z 178,A -21.5466,B 6.1123,C 0.3063,E1 6.2658,E2 473.8011} C_DIS
LIN {X 127.2399,Y -54.9357,Z 178,A -20.1514,B 6.1124,C 0.3031,E1 6.2673,E2 472.4085} C_DIS
LIN {X 128.7349,Y -51.3374,Z 178,A -18.6125,B 6.1126,C 0.3,E1 6.269,E2 470.8776} C_DIS
LIN {X 129.8134,Y -48.5429,Z 178,A -17.3342,B 6.1128,C 0.2959,E1 6.2702,E2 469.5929} C_DIS
LIN {X 131.2039,Y -44.6552,Z 178,A -15.7061,B 6.1129,C 0.2926,E1 6.2717,E2 467.9736} C_DIS
LIN {X 132.196,Y -41.6233,Z 178,A -13.8636,B 6.1135,C 0.2801,E1 6.2733,E2 466.0614} C_DIS
LIN {X 133.5324,Y -37.1094,Z 178,A -12.6878,B 6.1132,C 0.2878,E1 6.2742,E2 464.9845} C_DIS
LIN {X 134.2888,Y -34.2712,Z 178,A -11.3045,B 6.1135,C 0.2816,E1 6.2751,E2 463.5781} C_DIS
LIN {X 135.25,Y -30.2621,Z 178,A -9.6747,B 6.1136,C 0.278,E1 6.2762,E2 461.9566} C_DIS
LIN {X 135.9942,Y -26.7223,Z 178,A -8.243,B 6.1138,C 0.2749,E1 6.277,E2 460.5319} C_DIS
LIN {X 136.6169,Y -23.3262,Z 178,A -6.6577,B 6.1141,C 0.2682,E1 6.2777,E2 458.9249} C_DIS
LIN {X 137.3561,Y -18.4812,Z 178,A -4.953,B 6.1141,C 0.2679,E1 6.2784,E2 457.2601} C_DIS
LIN {X 137.8136,Y -14.679,Z 178,A -3.1054,B 6.1145,C 0.2589,E1 6.279,E2 455.3768} C_DIS
LIN {X 138.1682,Y -10.8729,Z 178,A -1.5892,B 6.1145,C 0.2555,E1 6.2793,E2 453.8678} C_DIS
LIN {X 138.4188,Y -6.9497,Z 178,A -0.1119,B 6.1147,C 0.2533,E1 6.2796,E2 452.4082} C_DIS
LIN {X 138.5478,Y -3.5574,Z 178,A 1.2745,B 6.1148,C 0.2496,E1 6.2796,E2 451.0229} C_DIS
LIN {X 138.5918,Y 0.7011,Z 178,A 3.0039,B 6.115,C 0.2451,E1 6.2797,E2 449.2962} C_DIS
LIN {X 138.5329,Y 4.0943,Z 178,A 4.4217,B 6.1152,C 0.2408,E1 6.2797,E2 447.8753} C_DIS
LIN {X 138.3587,Y 8.0701,Z 178,A 5.986,B 6.1153,C 0.2375,E1 6.2794,E2 446.3202} C_DIS
LIN {X 138.1007,Y 11.6726,Z 178,A 7.3664,B 6.1154,C 0.2352,E1 6.2791,E2 444.9532} C_DIS
LIN {X 137.4195,Y 17.9971,Z 178,A 10.3101,B 6.1159,C 0.2224,E1 6.2781,E2 441.967} C_DIS
LIN {X 136.8825,Y 21.7134,Z 178,A 11.4392,B 6.1158,C 0.2252,E1 6.2777,E2 440.8915} C_DIS
LIN {X 136.3857,Y 24.6373,Z 178,A 12.6669,B 6.1159,C 0.2217,E1 6.2771,E2 439.6627} C_DIS
LIN {X 135.269,Y 30.179,Z 178,A 14.9017,B 6.1161,C 0.2169,E1 6.2758,E2 437.4395} C_DIS
LIN {X 134.3726,Y 33.9411,Z 178,A 16.5777,B 6.1163,C 0.2111,E1 6.2747,E2 435.7525} C_DIS
LIN {X 133.4309,Y 37.4726,Z 178,A 18.003,B 6.1163,C 0.2084,E1 6.2736,E2 434.3372} C_DIS
LIN {X 132.4517,Y 40.7991,Z 178,A 19.3618,B 6.1165,C 0.2058,E1 6.2725,E2 432.9872} C_DIS
LIN {X 131.4168,Y 44.0184,Z 178,A 20.7962,B 6.1166,C 0.2014,E1 6.2713,E2 431.5472} C_DIS
LIN {X 130.0174,Y 47.9985,Z 178,A 23.8053,B 6.1174,C 0.1756,E1 6.2682,E2 428.3735} C_DIS
LIN {X 126.577,Y 56.4465,Z 178,A 25.9124,B 6.1169,C 0.1934,E1 6.2661,E2 426.4791} C_DIS
LIN {X 125.0787,Y 59.6929,Z 178,A 27.4028,B 6.1169,C 0.1893,E1 6.2643,E2 424.9863} C_DIS
LIN {X 124.0069,Y 61.8919,Z 178,A 28.611,B 6.1172,C 0.1835,E1 6.2628,E2 423.7526} C_DIS
LIN {X 122.4394,Y 64.9372,Z 178,A 30.0198,B 6.1172,C 0.1801,E1 6.261,E2 422.3441} C_DIS
LIN {X 116.8581,Y 74.5165,Z 178,A 34.2621,B 6.1174,C 0.1744,E1 6.2551,E2 418.1435} C_DIS
LIN {X 114.4604,Y 78.1498,Z 178,A 36.3289,B 6.1177,C 0.1658,E1 6.2518,E2 416.0422} C_DIS
LIN {X 112.0049,Y 81.6304,Z 178,A 38.0849,B 6.1177,C 0.1618,E1 6.2489,E2 414.2861} C_DIS
LIN {X 108.9182,Y 85.7048,Z 178,A 40.0916,B 6.1179,C 0.1587,E1 6.2455,E2 412.2922} C_DIS
LIN {X 106.4341,Y 88.7717,Z 178,A 41.7204,B 6.1179,C 0.1552,E1 6.2426,E2 410.6633} C_DIS
LIN {X 103.8457,Y 91.7853,Z 178,A 43.3402,B 6.118,C 0.152,E1 6.2397,E2 409.0458} C_DIS
Enddeposition()
END
